(* PLC project mtcs_services, Institute of Astronomy OntoManager 0.0.1 *)
(* stored: creationDateTime 2024-08-13T09:12:25.681669, modificationDateTime 2024-08-13T09:12:25.681669 *)

TYPE ServicesTimingTimeSource : (LOCAL_CLOCK := 0, PTP_IEEE_1588 := 1);
END_TYPE

TYPE ServicesMeteoId : (WIND_SPEED_MINIMUM := 0, WIND_SPEED_AVERAGE := 1, WIND_SPEED_MAXIMUM := 2, WIND_DIRECTION_MINIMUM := 3, WIND_DIRECTION_AVERAGE := 4, WIND_DIRECTION_MAXIMUM := 5, AIR_PRESSURE := 6, AIR_TEMPERATURE := 7, INTERNAL_TEMPERATURE := 8, RELATIVE_HUMIDITY := 9, RAIN_ACCUMULATION := 10, RAIN_DURATION := 11, RAIN_INTENSITY := 12, RAIN_PEAK_INTENSITY := 13, HAIL_ACCUMULATION := 14, HAIL_DURATION := 15, HAIL_PEAK_INTENSITY := 16, HAIL_INTENSITY := 17, HEATING_TEMPERATURE := 18, HEATING_VOLTAGE := 19, SUPPLY_VOLTAGE := 20, REFERENCE_VOLTAGE := 21);
END_TYPE

TYPE ServicesParts : STRUCT
  timing : ServicesTiming;  (* Timing service *)
  meteo : ServicesMeteo;  (* Meteo service *)
  west : ServicesWest;  (* West service *)
  chiller : ServicesChiller;  (* Chiller service *)
  io : ServicesIO;  (* I/O modules *)
  configManager : ConfigManager;  (* The config manager (to load/save/activate configuration data) *)
END_STRUCT;
END_TYPE

TYPE ServicesTimingParts : STRUCT
  serialInfo : ServicesTimingSerialInfo;  (* Info acquired by serial link *)
END_STRUCT;
END_TYPE

TYPE ServicesWestParts : STRUCT
  bus : ModbusRTUBus;  (* The shared Modbus RTU bus *)
  domeTemperature : ServicesWestController;  (* The West coparts.chillerMainController.parts.chillerMainControllerntroller at the dome to control the temperature *)
  firstFloorTemperature : ServicesWestController;  (* The West controller at the first floor to control the temperature *)
  pumpsRoomTemperature : ServicesWestController;  (* The West controller at the pumps room to control the temperature *)
  oilHeatExchangerTemperature : ServicesWestController;  (* The West controller at the heat exchanger to control the oil temperature *)
  serversRoomTemperature : ServicesWestController;  (* The West controller at the servers room to control the temperature *)
END_STRUCT;
END_TYPE

TYPE ServicesChillerParts : STRUCT
  bus : ModbusRTUBus;  (* The shared Modbus RTU bus *)
  chillerMainController : ServicesChillerController;  (* The Chiller controller to control the water temperature *)
END_STRUCT;
END_TYPE

TYPE ServicesIOParts : STRUCT
  coupler : EtherCatDevice;  (* Coupler *)
  slot1 : EtherCatDevice;  (* Slot 1 *)
  slot2 : EtherCatDevice;  (* Slot 2 *)
  slot3 : EtherCatDevice;  (* Slot 3 *)
  slot4 : EtherCatDevice;  (* Slot 4 *)
END_STRUCT;
END_TYPE

TYPE ServicesProcesses : STRUCT
  initialize : Process;  (* Start initializing *)
  lock : Process;  (* Lock the system *)
  unlock : Process;  (* Unlock the system *)
  changeOperatingState : ChangeOperatingStateProcess;  (* Change the operating state (e.g. AUTO, MANUAL, ...) *)
END_STRUCT;
END_TYPE

TYPE ServicesTimingProcesses : STRUCT

END_STRUCT;
END_TYPE

TYPE ServicesMeteoProcesses : STRUCT

END_STRUCT;
END_TYPE

TYPE ServicesWestControllerProcesses : STRUCT
  updateProcessVariables : Process;  (* Read process variables *)
  updateConfigVariables : Process;  (* Read config variables *)
  writeSetpoint : ChangeSetpointProcess;  (* Write the setpoint *)
  writeOffset : ChangeParameterProcess;  (* Set an internal offset to Process Value *)
  writeProportinalBand : ChangeParameterProcess;  (* Set the Proportinal band constant *)
  writeResetTime : ChangeParameterProcess;  (* Set the Integral time constant *)
  writeRate : ChangeParameterProcess;  (* Set the Derivative time constant *)
  switchToManual : Process;  (* Switch controller to Manual *)
  switchToAuto : Process;  (* Switch controller to Auto *)
  writeOutputPower : ChangeParameterProcess;  (* Set a specific output power *)
  writeConfigToController : Process;  (* Write saved config to Controller *)
END_STRUCT;
END_TYPE

TYPE ServicesWestProcesses : STRUCT
  changeOperatingState : ChangeOperatingStateProcess;  (* Change the operating state (e.g. AUTO, MANUAL, ...) *)
END_STRUCT;
END_TYPE

TYPE ServicesChillerControllerProcesses : STRUCT
  updateConfigVariables : Process;  (* Read the Config variables *)
  updateMeasureVariables : Process;  (* Read the Measurement variables *)
  updateAlarmRegisters : Process;  (* Read the Alarm registers *)
  writeSetpoint : ChangeSetpointProcess;  (* Write the setpoint *)
  switchChillerON : Process;  (* Switch ON the Chiller *)
  switchChillerOFF : Process;  (* Switch OFF the Chiller *)
  resetUnitController : Process;  (* Reset Unit controller of the Chiller *)
  resetAlarms : Process;  (* Reset all activated alarms *)
END_STRUCT;
END_TYPE

TYPE ServicesChillerProcesses : STRUCT
  changeOperatingState : ChangeOperatingStateProcess;  (* Change the operating state (e.g. AUTO, MANUAL, ...) *)
END_STRUCT;
END_TYPE

TYPE ServicesStatuses : STRUCT
  initializationStatus : InitializationStatus;
  healthStatus : HealthStatus;
  busyStatus : BusyStatus;
  operatingStatus : OperatingStatus;
END_STRUCT;
END_TYPE

TYPE ServicesTimingStatuses : STRUCT
  healthStatus : HealthStatus;
END_STRUCT;
END_TYPE

TYPE ServicesTimingSerialInfoStatuses : STRUCT
  portHealthStatus : HealthStatus;
  transmissionHealthStatus : HealthStatus;
  checksumHealthStatus : HealthStatus;
  healthStatus : HealthStatus;
END_STRUCT;
END_TYPE

TYPE ServicesMeteoMeasurementStatuses : STRUCT
  enabledStatus : EnabledStatus;  (* Is the temperature being measured? *)
  healthStatus : HealthStatus;  (* Is the data valid and within range? *)
  alarmStatus : HiHiLoLoAlarmStatus;  (* Alarm status *)
END_STRUCT;
END_TYPE

TYPE ServicesMeteoStatuses : STRUCT
  meteoHealthStatus : HealthStatus;
  healthStatus : HealthStatus;
END_STRUCT;
END_TYPE

TYPE ServicesWestControllerStatuses : STRUCT
  healthStatus : HealthStatus;  (* Is the data valid and within range? *)
  alarmStatus : HiHiLoLoAlarmStatus;  (* Alarm status *)
END_STRUCT;
END_TYPE

TYPE ServicesWestStatuses : STRUCT
  healthStatus : HealthStatus;  (* Are the WESTs in healthy state (good) or not (bad) *)
  operatingStatus : OperatingStatus;  (* Are the WESTs being polled (auto) or not (manual)? *)
END_STRUCT;
END_TYPE

TYPE ServicesChillerControllerStatuses : STRUCT
  healthStatus : HealthStatus;  (* Is the data valid and within range? *)
  alarmStatusWatertemperature : HiHiLoLoAlarmStatus;  (* Alarm status about Water temperature *)
  alarmStatusWaterPumpSupervisor : HiHiLoLoAlarmStatus;  (* Alarm status about WaterPump supervisor *)
END_STRUCT;
END_TYPE

TYPE ServicesChillerStatuses : STRUCT
  healthStatus : HealthStatus;  (* Is the Chiller in healthy state (good) or not (bad) *)
  operatingStatus : OperatingStatus;  (* Is the Chiller being polled (auto) or not (manual)? *)
END_STRUCT;
END_TYPE

TYPE ServicesIOStatuses : STRUCT
  healthStatus : HealthStatus;  (* Is the I/O in a healthy state? *)
END_STRUCT;
END_TYPE

TYPE ServicesTimingConfig : STRUCT
  leapSeconds : INT;  (* Number of leap seconds, so that UTC = TAI + this value. See ftp://maia.usno.navy.mil/ser7/tai-utc.dat for the latest number. *)
  dut : LREAL;  (* Delta UT (= UT1 - UTC). Put to 0.0 to ignore. *)
  alwaysUseLocalClock : BOOL;  (* If TRUE, then the local clock (source=LOCAL_CLOCK) will be used even if an external (more accurate!) clock is available *)
  ignoreSerialError : BOOL;  (* Don't show the Servicestiming status as ERROR in case the serial link fails *)
END_STRUCT;
END_TYPE

TYPE ServicesMeteoConfig : STRUCT
  enableWeatherMonitoring : BOOL;  (* Enable weather monitoring and emergency closing *)
  wetLimit : LREAL;  (* Wet if (rainIntensity+hailIntrelaensity)>wetLimit *)
  windSpeedMinimum : MeasurementConfig;  (* Config for the wind speed minimum *)
  windSpeedAverage : MeasurementConfig;  (* Config for the wind speed average *)
  windSpeedMaximum : MeasurementConfig;  (* Config for the wind speed maximum *)
  windDirectionMinimum : MeasurementConfig;  (* Config for the wind direction minimum *)
  windDirectionAverage : MeasurementConfig;  (* Config for the wind direction average *)
  windDirectionMaximum : MeasurementConfig;  (* Config for the wind direction maximum *)
  airPressure : MeasurementConfig;  (* Config for the air pressure *)
  airTemperature : MeasurementConfig;  (* Config for the air temperature *)
  internalTemperature : MeasurementConfig;  (* Config for the internal temperature *)
  relativeHumidity : MeasurementConfig;  (* Config for the relative humidity *)
  rainAccumulation : MeasurementConfig;  (* Config for the rain accumulation *)
  rainDuration : MeasurementConfig;  (* Config for the rain duration *)
  rainIntensity : MeasurementConfig;  (* Config for the rain intensity *)
  rainPeakIntensity : MeasurementConfig;  (* Config for the rain peak intensity *)
  hailAccumulation : MeasurementConfig;  (* Config for the hail accumulation *)
  hailDuration : MeasurementConfig;  (* Config for the hail duration *)
  hailIntensity : MeasurementConfig;  (* Config for the hail intensity *)
  hailPeakIntensity : MeasurementConfig;  (* Config for the hail peak intensity *)
  heatingTemperature : MeasurementConfig;  (* Config for the heating temperature *)
  heatingVoltage : MeasurementConfig;  (* Config for the heating voltage *)
  supplyVoltage : MeasurementConfig;  (* Config for the supply voltage *)
  referenceVoltage : MeasurementConfig;  (* Config for the 3.5 V reference voltage *)
END_STRUCT;
END_TYPE

TYPE ServicesWestTemperatureTimeConfig : STRUCT
  enable : BOOL;  (* Enable this time (TRUE) or not (FALSE) *)
  hour : LREAL;  (* The time to change the setpoint, as decimal hour (e.g. 9.5 = 9:30 am) *)
  offset : LREAL;  (* Setpoint = air temperature of meteo station + this offset (in degrees celsius) *)
END_STRUCT;
END_TYPE

TYPE ServicesWestTemperatureUpdateConfig : STRUCT
  time0 : ServicesWestTemperatureTimeConfig;  (* Time config 0 *)
  time1 : ServicesWestTemperatureTimeConfig;  (* Time config 1 *)
  time2 : ServicesWestTemperatureTimeConfig;  (* Time config 2 *)
  time3 : ServicesWestTemperatureTimeConfig;  (* Time config 3 *)
  time4 : ServicesWestTemperatureTimeConfig;  (* Time config 4 *)
END_STRUCT;
END_TYPE

TYPE ServicesWestParametersAddressesConfig : STRUCT
  communicationWriteStatus : UINT := 1;  (* Communication Write Status *)
  manualControl : UINT := 2;  (* Manual control *)
  selfTune : UINT := 3;  (* Activate SelfTune *)
  preTune : UINT := 4;  (* Activate PreTune *)
  alarm1Status : UINT := 5;  (* Alarm 1 status *)
  alarm2Status : UINT := 6;  (* Alarm 2 status *)
  setpointRampling : UINT := 7;  (* Setpoint ramping *)
  loopAlarmStatus : UINT := 10;  (* Loop alarm status *)
  loopAlarm : UINT := 12;  (* Loop alarm *)
  digitalInput2 : UINT := 13;  (* State Option B digital input *)
  processVariable : UINT := 1;  (* Process Variable *)
  setpoint : UINT := 2;  (* Setpoint *)
  outputPower : UINT := 3;  (* Power percentage *)
  desviation : UINT := 4;  (* Difference ProcessVariable and Setpoint *)
  primaryProportionalBand : UINT := 6;  (* Primary Proportional band PB *)
  directActing : UINT := 7;  (* Direct reverse acting *)
  resetTime : UINT := 8;  (* Reset Time. Integral time constant *)
  rate : UINT := 9;  (* Rate. Derivative time constant *)
  output1ClycleTime : UINT := 10;  (* Output 1 cycle time in seconds *)
  scaleRangeLowerLimit : UINT := 11;  (* Lower Limit of input range *)
  scaleRangeUpperLimit : UINT := 12;  (* Upper Limit of input range *)
  alarm1Value : UINT := 13;  (* Alarm 1 active at this level *)
  alarm2Value : UINT := 14;  (* Alarm 2 active at this level *)
  manualReset : UINT := 15;  (* Bias value in percentage *)
  deadbandOverlap : UINT := 16;  (* Deadband and Overlap percentage *)
  onOffDiferential : UINT := 17;  (* Input span for ON/OFF differential *)
  decimalPointPosition : UINT := 18;  (* Decimal point position *)
  output2ClycleTime : UINT := 19;  (* Output 2 cycle time in seconds *)
  primaryOutputPowerLimit : UINT := 20;  (* Safety power limit in porcentage *)
  actualSetpoint : UINT := 21;  (* Current Setpoint value (ramping) *)
  setpointUpperLimit : UINT := 22;  (* Setpoint upper limit *)
  setpointLowerLimit : UINT := 23;  (* Setpoint lower limit *)
  setpointRampRate : UINT := 24;  (* Setpoint ramp rate *)
  inputFilterTimeContant : UINT := 25;  (* Input Filter time contant *)
  processValueOffset : UINT := 26;  (* Process Value offset *)
  alarm1Hysteresis : UINT := 32;  (* Alarm 1 hysteresis in percentage *)
  alarm2Hysteresis : UINT := 33;  (* Alarm 2 hysteresis in percentage *)
END_STRUCT;
END_TYPE

TYPE ServicesWestControllerVariables : STRUCT
  setpoint : LREAL;  (* Setpoint *)
  defaultSetpoint : LREAL;  (* Default setpoint *)
  minSetpoint : LREAL;  (* Minimun setpoint *)
  maxSetpoint : LREAL;  (* Maximal setpoint *)
  processValueOffset : LREAL;  (* Offset process varible *)
  differentialOnOff : LREAL;  (* On/Off differential *)
  alarmValue : LREAL;  (* Alarm value *)
  inputFilterTimeConstant : LREAL;  (* Input filter time constant *)
  cycleTime : LREAL;  (* Cycle time for control loop *)
  proportionalBand : UINT;  (* Proportional constant *)
  resetTime : UINT;  (* Integral time constant *)
  rate : UINT;  (* Dervative time constant *)
END_STRUCT;
END_TYPE

TYPE ServicesWestControllerConfig : STRUCT
  unitID : USINT;  (* The address or UnitID of the controller *)
  update : BOOL;  (* True to automatically update the setpoint *)
  warningMessage : STRING;  (* A warning message (empty = not shown) *)
  measurement : MeasurementConfig;  (* The measurement config *)
  variables : ServicesWestControllerVariables;  (* Configuration parameters *)
END_STRUCT;
END_TYPE

TYPE ServicesWestConfig : STRUCT
  updateProcessVariables : BOOL;  (* True to automatically update process variables *)
  updateVariablesPollingInterval : LREAL;  (* Time between bus reads in seconds *)
  domeTempControl : BOOL;  (* True to automatically update dome temperatures *)
  domeTempCycleTime : LREAL;  (* Time between bus checks in seconds *)
  hydraulicsTempControl : BOOL;  (* True to enable PID controller for hydraulics temperatures *)
  hydraulicsTempCycleTime : LREAL;  (* Cycle time for PID Controller in seconds *)
  hydraulicsProportionalConstantKP : LREAL;  (* Proportional constant (Kp) for PID Controller *)
  hydraulicsIntegralConstantTn : LREAL;  (* Integral constant (Tn) for PID Controller in seconds *)
  domeTemperature : ServicesWestControllerConfig;  (* The address of the Dome temperature controller *)
  firstFloorTemperature : ServicesWestControllerConfig;  (* The address of the first floor temperature controller *)
  pumpsRoomTemperature : ServicesWestControllerConfig;  (* The address of the pumps room temperature controller *)
  oilHeatExchangerTemperature : ServicesWestControllerConfig;  (* The address of the oil heat exchanger temperature controller *)
  serversRoomTemperature : ServicesWestControllerConfig;  (* The address of the servers room temperature controller *)
  parameterAddresses : ServicesWestParametersAddressesConfig;  (* Config about Modbus parameters addresses *)
  temperatureUpdate : ServicesWestTemperatureUpdateConfig;  (* The config for the temperature setpoint *)
END_STRUCT;
END_TYPE

TYPE ServicesChillerControllerParameterAddresses : STRUCT
  waterTankTemperature : UINT := 258;  (* Water tank temperature *)
  highPressureCircuit1 : UINT := 260;  (* High pressure of circuit 1 *)
  highPressureCircuit2 : UINT := 262;  (* High pressure of circuit 2 *)
  chillerCurrentInput : UINT := 264;  (* Chiller current input *)
  waterPumpCurrentInput : UINT := 266;  (* Water pump current input *)
  evaporatorOutTemp1 : UINT := 268;  (* Evaporator out temperature 1 *)
  evaporatorOutTemp2 : UINT := 270;  (* Evaporator out temperature 2 *)
  ambientTemperature : UINT := 272;  (* Ambient temperature *)
  waterPumpChassisTemp : UINT := 274;  (* Water Pump chassis temperature *)
  digitalInputStatus1 : UINT := 512;  (* Flow switch status *)
  digitalInputStatus2 : UINT := 513;  (* Digital input status 2 *)
  digitalInputStatus3 : UINT := 514;  (* Digital input status 3 *)
  digitalInputStatus4 : UINT := 515;  (* Digital input status 4 *)
  setpoint : UINT := 768;  (* Setpoint parameter address *)
  minSetpoint : UINT := 769;  (* Minimal Setpoint parameter address *)
  maxSetpoint : UINT := 770;  (* Maximal Setpoint parameter address *)
  trippingBand : UINT := 774;  (* Tripping Band parameter address *)
  unitStatus : UINT := 1280;  (* Unit Status parameter address *)
  unitControllerReset : UINT := 1282;  (* Unit Controlelr reset parameter address *)
  relayOutputStatus1 : UINT := 2048;  (* Relay output status 1 *)
  relayOutputStatus2 : UINT := 2049;  (* Relay output status 2 *)
  relayOutputStatus3 : UINT := 2050;  (* Relay output status 3 *)
  relayOutputStatus4 : UINT := 2051;  (* Relay output status 4 *)
  relayOutputStatus5 : UINT := 2052;  (* Relay output status 5 *)
  relayOutputStatus6 : UINT := 2053;  (* Relay output status 6 *)
  relayOutputStatus7 : UINT := 2054;  (* Relay output status 7 *)
  AnalogOutputStatus1 : UINT := 2304;  (* Fan Condenser1 Output *)
  AnalogOutputStatus2 : UINT := 2306;  (* Fan Condenser2 Output *)
  alarmStatus1 : UINT := 3328;  (* Alarm status 1 *)
  alarmStatus2 : UINT := 3329;  (* Alarm status 2 *)
  alarmStatus3 : UINT := 3330;  (* Alarm status 3 *)
  alarmStatus6 : UINT := 3333;  (* Alarm status 6 *)
  alarmStatus7 : UINT := 3334;  (* Alarm status 7 *)
  alarmStatus10 : UINT := 3337;  (* Alarm status 10 *)
  alarmStatus11 : UINT := 3338;  (* Alarm status 11 *)
  hoursCompressor1 : UINT := 3584;  (* Operation hours of compressor 1 *)
  hoursCompressor2 : UINT := 3585;  (* Operation hours of compressor 2 *)
  hoursCompressor3 : UINT := 3586;  (* Operation hours of compressor 3 *)
  hoursCompressor4 : UINT := 3587;  (* Operation hours of compressor 4 *)
  hoursPump : UINT := 3590;  (* Operation hours of water pump *)
  alarmOilCompressor1 : UINT := 3840;  (* Alarm oil Compressor 1 *)
  alarmOilCompressor2 : UINT := 3841;  (* Alarm oil Compressor 2 *)
  alarmOilCompressor3 : UINT := 3842;  (* Alarm oil Compressor 3 *)
  alarmOilCompressor4 : UINT := 3843;  (* Alarm oil Compressor 4 *)
  alarmFanOverload : UINT := 3846;  (* Alarm fan overload *)
  alarmColdSideFlowSwitch : UINT := 3847;  (* Alarm cold side flow switch *)
  alarmHotSideFlowSwitch : UINT := 3848;  (* Alarm hot side flow switch *)
  alarmCirc1LowTempPressDI : UINT := 3849;  (* Alarm circuit 1 low temppress DI *)
  alarmCirc2LowTempPressDI : UINT := 3850;  (* Alarm circuit 2 low temppress DI *)
  alarmCirc1LowTempPressPB : UINT := 3851;  (* Alarm circuit 1 low temppress PB *)
  alarmCirc2LowTempPressPB : UINT := 3852;  (* Alarm circuit 2 low temppress PB *)
END_STRUCT;
END_TYPE

TYPE ServicesChillerControllerAlarmStatus1 : STRUCT
  bit0 : STRING := 'PROBE8 (EVAP2. WATER TEMPERATURE)';
  bit1 : STRING := 'PROBE9 (AMBIENT TEMPERATURE)';
  bit2 : STRING := 'PROBE10 (NOT USED)';
  bit3 : STRING := 'PROBE11 (NOT USED)';
  bit4 : STRING := 'PROBE12 (NOT USED)';
  bit5 : STRING := 'COMPRESSOR1 MAINTENANCE';
  bit6 : STRING := 'COMPRESSOR2 MAINTENANCE';
  bit7 : STRING := 'COMPRESSOR3 MAINTENANCE';
  bit8 : STRING := 'ALARM NOT DEFINED';
  bit9 : STRING := 'PROBE1 (NOT USED)';
  bit10 : STRING := 'PROBE2 (TANK. WATER TEMPERATURE)';
  bit11 : STRING := 'PROBE3 (HIGH PRESSURE CRIC1)';
  bit12 : STRING := 'PROBE4 (HIGH PRESSURE CRIC2)';
  bit13 : STRING := 'PROBE5 (NOT USED)';
  bit14 : STRING := 'PROBE6 (NOT USED)';
  bit15 : STRING := 'PROBE7 (EVAP1. WATER TEMPERATURE)';
END_STRUCT;
END_TYPE

TYPE ServicesChillerControllerAlarmStatus2 : STRUCT
  bit0 : STRING := 'ALARM NOT DEFINED';
  bit1 : STRING := 'ALARM NOT DEFINED';
  bit2 : STRING := 'ALARM NOT DEFINED';
  bit3 : STRING := 'ALARM NOT DEFINED';
  bit4 : STRING := 'ALARM NOT DEFINED';
  bit5 : STRING := 'ALARM NOT DEFINED';
  bit6 : STRING := 'ALARM NOT DEFINED';
  bit7 : STRING := 'ALARM NOT DEFINED';
  bit8 : STRING := 'COMPRESSOR4 MAINTENANCE';
  bit9 : STRING := 'ALARM NOT DEFINED';
  bit10 : STRING := 'ALARM NOT DEFINED';
  bit11 : STRING := 'PUMP/DELIVERY FAN MAINTENANCE';
  bit12 : STRING := 'EVAPORATOR2 PUMP MAINTENANCE';
  bit13 : STRING := 'CONDENSER1 PUMP MAINTENANCE';
  bit14 : STRING := 'CONDENSER2 PUMP MAINTENANCE';
  bit15 : STRING := 'ALARM NOT DEFINED';
END_STRUCT;
END_TYPE

TYPE ServicesChillerControllerAlarmStatus3 : STRUCT
  bit0 : STRING := 'ALARM NOT DEFINED';
  bit1 : STRING := 'ALARM NOT DEFINED';
  bit2 : STRING := 'ALARM NOT DEFINED';
  bit3 : STRING := 'ALARM NOT DEFINED';
  bit4 : STRING := 'ALARM NOT DEFINED';
  bit5 : STRING := 'ALARM NOT DEFINED';
  bit6 : STRING := 'ALARM NOT DEFINED';
  bit7 : STRING := 'ALARM NOT DEFINED';
  bit8 : STRING := 'CIRCUIT1 DEFROST';
  bit9 : STRING := 'CIRCUIT2 DEFROST';
  bit10 : STRING := 'NETWORK FREQUENCY';
  bit11 : STRING := 'LOW INLET AIR TEMPERATURE';
  bit12 : STRING := 'ALARM NOT DEFINED';
  bit13 : STRING := 'ALARM NOT DEFINED';
  bit14 : STRING := 'EVAPORATOR LOW OUTLET TEMPERATURE';
  bit15 : STRING := 'EVAPORATOR HIGH OUTLET TEMPERATURE';
END_STRUCT;
END_TYPE

TYPE ServicesChillerControllerAlarmStatus6 : STRUCT
  bit0 : STRING := 'COMPRESSOR1 THERMAL OVERLOAD';
  bit1 : STRING := 'COMPRESSOR2 THERMAL OVERLOAD';
  bit2 : STRING := 'COMPRESSOR3 THERMAL OVERLOAD';
  bit3 : STRING := 'COMPRESSOR4 THERMAL OVERLOAD';
  bit4 : STRING := 'ALARM NOT DEFINED';
  bit5 : STRING := 'ALARM NOT DEFINED';
  bit6 : STRING := 'CIRC1 COND. FAN THERMAL OVERLOAD';
  bit7 : STRING := 'CIRC2 COND. FAN THERMAL OVERLOAD';
  bit8 : STRING := 'ALARM NOT DEFINED';
  bit9 : STRING := 'ALARM NOT DEFINED';
  bit10 : STRING := 'COMPRESSOR1 HIGH PRESSURE';
  bit11 : STRING := 'COMPRESSOR2 HIGH PRESSURE';
  bit12 : STRING := 'COMPRESSOR3 HIGH PRESSURE';
  bit13 : STRING := 'COMPRESSOR4 HIGH PRESSURE';
  bit14 : STRING := 'ALARM NOT DEFINED';
  bit15 : STRING := 'ALARM NOT DEFINED';
END_STRUCT;
END_TYPE

TYPE ServicesChillerControllerAlarmStatus7 : STRUCT
  bit0 : STRING := 'ALARM NOT DEFINED';
  bit1 : STRING := 'ALARM NOT DEFINED';
  bit2 : STRING := 'ALARM NOT DEFINED';
  bit3 : STRING := 'ALARM NOT DEFINED';
  bit4 : STRING := 'ALARM NOT DEFINED';
  bit5 : STRING := 'ALARM NOT DEFINED';
  bit6 : STRING := 'ALARM NOT DEFINED';
  bit7 : STRING := 'ALARM NOT DEFINED';
  bit8 : STRING := 'EVAP1 WATER PUMP THERMAL OVERLOAD';
  bit9 : STRING := 'EVAP2 WATER PUMP THERMAL OVERLOAD';
  bit10 : STRING := 'COND1 PUMP THERMAL OVERLOAD';
  bit11 : STRING := 'COND2 PUMP THERMAL OVERLOAD';
  bit12 : STRING := 'CIRC1 HIGH PRESSURE SWITCH TRIPPED';
  bit13 : STRING := 'CIRC2 HIGH PRESSURE SWITCH TRIPPED';
  bit14 : STRING := 'CIRC1 HIGH PRESSURE PROBE';
  bit15 : STRING := 'CIRC2 HIGH PRESSURE PROBE';
END_STRUCT;
END_TYPE

TYPE ServicesChillerControllerAlarmStatus10 : STRUCT
  bit0 : STRING := 'HOT SIDE FLOW SWITCH';
  bit1 : STRING := 'CIC1 LOW PRESSURE SWITCH';
  bit2 : STRING := 'CIC2 LOW PRESSURE SWITCH';
  bit3 : STRING := 'CIC1 LOW PRESSURE PROBE';
  bit4 : STRING := 'CIC2 LOW PRESSURE PROBE';
  bit5 : STRING := 'CIRC1 PUMP-DOWN AT STARTUP';
  bit6 : STRING := 'CIRC2 PUMP-DOWN AT STARTUP';
  bit7 : STRING := 'CIRC1 PUMP-DOWN AT SHUTDOWN';
  bit8 : STRING := 'COMPRESSOR1 OIL';
  bit9 : STRING := 'COMPRESSOR2 OIL';
  bit10 : STRING := 'COMPRESSOR3 OIL';
  bit11 : STRING := 'COMPRESSOR4 OIL';
  bit12 : STRING := 'ALARM NOT DEFINED';
  bit13 : STRING := 'ALARM NOT DEFINED';
  bit14 : STRING := 'DELIVERY FAN THERMAL OVERLOAD';
  bit15 : STRING := 'COLD SIDE FLOW SWITCH';
END_STRUCT;
END_TYPE

TYPE ServicesChillerControllerAlarmStatus11 : STRUCT
  bit0 : STRING := 'COMPRESSOR4 DISCHARGE HIGH TEMPERATURE';
  bit1 : STRING := 'ALARM NOT DEFINED';
  bit2 : STRING := 'ALARM NOT DEFINED';
  bit3 : STRING := 'GENERAL ALARM FROM DIGITAL INPUT';
  bit4 : STRING := 'ALARM NOT DEFINED';
  bit5 : STRING := 'ALARM NOT DEFINED';
  bit6 : STRING := 'ALARM NOT DEFINED';
  bit7 : STRING := 'ALARM NOT DEFINED';
  bit8 : STRING := 'CIRC2 PUMP-DOWN AT SHUTDOWN';
  bit9 : STRING := 'CIRC1 CHILLER ANTI-FREEZE';
  bit10 : STRING := 'CIRC2 CHILLER ANTI-FREEZE';
  bit11 : STRING := 'CIRC1 PUMP ANTI-FREEZE';
  bit12 : STRING := 'CIRC2 PUMP ANTI-FREEZE';
  bit13 : STRING := 'COMPRESSOR1 DISCHARGE HIGH TEMPERATURE';
  bit14 : STRING := 'COMPRESSOR2 DISCHARGE HIGH TEMPERATURE';
  bit15 : STRING := 'COMPRESSOR3 DISCHARGE HIGH TEMPERATURE';
END_STRUCT;
END_TYPE

TYPE ServicesChillerControllerBitwiseConfig : STRUCT
  statusOnMask : UINT := 768;  (* Word check if Chiller is ON *)
  switchOnMask : UINT := 1028;  (* Word to switch ON the Chiller *)
  switchOffMask : UINT := 1;  (* Word to switch OFF the Chiller *)
  resetUnitMask : UINT := 128;  (* Word to reset controller Unit *)
  resetAlarmMask : UINT := 4112;  (* Word to reset Alarm *)
  flowSwitchMask : UINT := 2048;  (* Word to check if Flow switch is ON *)
  alarmOnMask : UINT := 257;  (* Word to check if Alarm relay is ON *)
  waterPumpOnMask : UINT := 514;  (* Word to check if water Pump relay is ON *)
  compressor1Mask : UINT := 8224;  (* Word to check if Compressor1 is ON *)
  compressor2Mask : UINT := 4112;  (* Word to check if Compressor2 is ON *)
  compressor3Mask : UINT := 2056;  (* Word to check if Compressor3 is ON *)
  compressor4Mask : UINT := 1028;  (* Word to check if Compressor4 is ON *)
  bit0 : UINT := 1;  (* Word mask to check bit0 *)
  bit1 : UINT := 2;  (* Word mask to check bit1 *)
  bit2 : UINT := 4;  (* Word mask to check bit2 *)
  bit3 : UINT := 8;  (* Word mask to check bit3 *)
  bit4 : UINT := 16;  (* Word mask to check bit4 *)
  bit5 : UINT := 32;  (* Word mask to check bit5 *)
  bit6 : UINT := 64;  (* Word mask to check bit6 *)
  bit7 : UINT := 128;  (* Word mask to check bit7 *)
  bit8 : UINT := 256;  (* Word mask to check bit8 *)
  bit9 : UINT := 512;  (* Word mask to check bit9 *)
  bit10 : UINT := 1024;  (* Word mask to check bit10 *)
  bit11 : UINT := 2048;  (* Word mask to check bit11 *)
  bit12 : UINT := 4096;  (* Word mask to check bit12 *)
  bit13 : UINT := 8192;  (* Word mask to check bit13 *)
  bit14 : UINT := 16384;  (* Word mask to check bit14 *)
  bit15 : UINT := 32768;  (* Word mask to check bit15 *)
END_STRUCT;
END_TYPE

TYPE ServicesChillerControllerAlarmStatusRegisters : STRUCT
  AlarmStatus1 : ServicesChillerControllerAlarmStatus1;  (* Alarm indicators at AlarmStatus1 register *)
  AlarmStatus2 : ServicesChillerControllerAlarmStatus2;  (* Alarm indicators at AlarmStatus2 register *)
  AlarmStatus3 : ServicesChillerControllerAlarmStatus3;  (* Alarm indicators at AlarmStatus3 register *)
  AlarmStatus6 : ServicesChillerControllerAlarmStatus6;  (* Alarm indicators at AlarmStatus6 register *)
  AlarmStatus7 : ServicesChillerControllerAlarmStatus7;  (* Alarm indicators at AlarmStatus7 register *)
  AlarmStatus10 : ServicesChillerControllerAlarmStatus10;  (* Alarm indicators at AlarmStatus10 register *)
  AlarmStatus11 : ServicesChillerControllerAlarmStatus11;  (* Alarm indicators at AlarmStatus11 register *)
END_STRUCT;
END_TYPE

TYPE ServicesChillerControllerVariables : STRUCT
  setpoint : LREAL;  (* Setpoint *)
  minSetpoint : LREAL;  (* Minimun setpoint *)
  maxSetpoint : LREAL;  (* Maximal setpoint *)
  trippingBand : LREAL;  (* Tripping band *)
END_STRUCT;
END_TYPE

TYPE ServicesChillerControllerConfig : STRUCT
  unitID : USINT;  (* The address or UnitID of the controller *)
  waterTankTemperatureMeasurement : MeasurementConfig;  (* The WaterTank measurement config *)
  warningMessageWaterTemperatureMeasurement : STRING;  (* A warning message (empty = not shown) *)
  waterPumpSupervisorMeasurement : MeasurementConfig;  (* The WaterPump supervisor measurement config *)
  messageWaterPumpSupervisorMeasurement : STRING;  (* A message to be shown on config tab *)
  warningMessageWaterPumpSupervisorMeasurement : STRING;  (* A warning message (empty = not shown) *)
  parameterAddresses : ServicesChillerControllerParameterAddresses;  (* Config about Modbus parameters addresses *)
  variables : ServicesChillerControllerVariables;  (* Config value for some parameters *)
  alarmRegisters : ServicesChillerControllerAlarmStatusRegisters;  (* Config about Alarm statuses registers *)
  bitwise : ServicesChillerControllerBitwiseConfig;  (* Config about words and masks for bitwise actions *)
END_STRUCT;
END_TYPE

TYPE ServicesChillerConfig : STRUCT
  updateSetpoint : BOOL;  (* True to automatically update the setpoint *)
  temperatureToChangeSetpoint : LREAL;  (* Temperature to change Setpoint *)
  summerSetpoint : LREAL;  (* Temperature setpoint for summer *)
  winterSetpoint : LREAL;  (* Temperature setpoint for winter *)
  offsetSetpoint : LREAL;  (* Setpoint = air temperature of meteo station + this offset (in degrees celsius) *)
  updateSetpointInterval : LREAL;  (* Time interval to check ambient/setpoint temperature in seconds *)
  updateVariables : BOOL;  (* True to automatically update the setpoint *)
  pollingMeasuresInterval : LREAL;  (* Time between bus measurement reads in seconds *)
  pollingConfigInterval : LREAL;  (* Time between bus config variables reads in seconds *)
  pollingAlarmsInterval : LREAL;  (* Time between bus alarm registers reads in seconds *)
  chillerMainController : ServicesChillerControllerConfig;  (* The Chiller controller config *)
END_STRUCT;
END_TYPE

TYPE ServicesConfig : STRUCT
  timing : ServicesTimingConfig;  (* Timing config *)
  meteo : ServicesMeteoConfig;  (* Meteo config *)
  west : ServicesWestConfig;  (* West config *)
  chiller : ServicesChillerConfig;  (* Chiller config *)
END_STRUCT;
END_TYPE

FUNCTION_BLOCK SM_Services
  VAR_INPUT
    {attribute 'OPC.UA.DA' := '1'}
    {attribute 'OPC.UA.DA.Access' := '1'}
    editableConfig : ServicesConfig;  (* Editable configuration of the Services subsystem *)
  END_VAR
  VAR_OUTPUT
    {attribute 'OPC.UA.DA' := '1'}
    {attribute 'OPC.UA.DA.Access' := '1'}
    actualStatus : STRING;  (* Current status description *)
    previousStatus : STRING;  (* Previous status description *)
    {attribute 'OPC.UA.DA' := '1'}
    {attribute 'OPC.UA.DA.Access' := '1'}
    config : ServicesConfig;  (* Active configuration of the Services subsystem *)
    statuses : ServicesStatuses;  (* Statuses of the state machine *)
    parts : ServicesParts;  (* Parts of the state machine *)
    processes : ServicesProcesses;  (* Processes of the state machine *)
  END_VAR
  VAR_IN_OUT
    {attribute 'OPC.UA.DA' := '0'}
    operatorStatus : OperatorStatus;  (* Shared operator status *)
    {attribute 'OPC.UA.DA' := '0'}
    domeApertureStatus : ApertureStatus;  (* Is the dome open or closed? *)
  END_VAR

            parts.timing(
    operatorStatus := operatorStatus,
    config := config.timing);
parts.meteo( config := config.meteo );
parts.west(
    operatorStatus := operatorStatus,
    config := config.west,
    airTemperature := parts.meteo.airTemperature,
    domeApertureStatus := domeApertureStatus);
parts.chiller(
    operatorStatus := operatorStatus,
    config := config.chiller,
    airTemperature := parts.meteo.airTemperature);
parts.io();
parts.configManager( isEnabled := operatorStatus.tech );
statuses.initializationStatus();
statuses.healthStatus(
    isGood := parts.timing.statuses.healthStatus.isGood AND (parts.meteo.statuses.healthStatus.isGood AND (parts.west.statuses.healthStatus.isGood AND (parts.chiller.statuses.healthStatus.isGood AND parts.io.statuses.healthStatus.isGood))),
    hasWarning := parts.timing.statuses.healthStatus.hasWarning OR (parts.meteo.statuses.healthStatus.hasWarning OR (parts.west.statuses.healthStatus.hasWarning OR (parts.chiller.statuses.healthStatus.hasWarning OR parts.io.statuses.healthStatus.hasWarning))));
statuses.busyStatus( isBusy := statuses.initializationStatus.initializing );
statuses.operatingStatus( superState := statuses.initializationStatus.initialized );
processes.initialize( isEnabled := statuses.initializationStatus.shutdown OR (statuses.initializationStatus.initializingFailed OR statuses.initializationStatus.initialized) );
processes.lock( isEnabled := operatorStatus.tech AND statuses.initializationStatus.initialized );
processes.unlock( isEnabled := operatorStatus.tech AND statuses.initializationStatus.locked );
processes.changeOperatingState( isEnabled := FALSE );

          

{attribute 'TcRpcEnable' := '1'}
METHOD initialize : RequestResults
                  initialize := THIS^.processes.initialize.request();

                
END_METHOD

{attribute 'TcRpcEnable' := '1'}
METHOD lock : RequestResults
                  lock := THIS^.processes.lock.request();

                
END_METHOD

{attribute 'TcRpcEnable' := '1'}
METHOD unlock : RequestResults
                  unlock := THIS^.processes.unlock.request();

                
END_METHOD

{attribute 'TcRpcEnable' := '1'}
METHOD changeOperatingState : RequestResults
  VAR_INPUT
    state : OperatingStates;
  END_VAR
                  changeOperatingState := THIS^.processes.changeOperatingState.request( state := state );

                
END_METHOD

{attribute 'TcRpcEnable' := '1'}
METHOD _log : BOOL
  VAR_INPUT
    name : STRING;  (* Name of this function block instance *)
  END_VAR
  VAR_IN_OUT
    buffer : LogBuffer;  (* Buffer to write all logging to *)
  END_VAR
  VAR
    subBuffer : LogBuffer;  (* Temporary buffer to write logging by parts (sub-statemachines) to *)
  END_VAR
                  THIS^.parts.timing._log(
    name := 'timing',
    buffer := subBuffer);
THIS^.parts.meteo._log(
    name := 'meteo',
    buffer := subBuffer);
THIS^.parts.west._log(
    name := 'west',
    buffer := subBuffer);
THIS^.parts.chiller._log(
    name := 'chiller',
    buffer := subBuffer);
THIS^.parts.io._log(
    name := 'io',
    buffer := subBuffer);
THIS^.parts.configManager._log(
    name := 'configManager',
    buffer := subBuffer);
THIS^.processes.initialize._log(
    name := 'processes.initialize',
    buffer := subBuffer);
THIS^.processes.lock._log(
    name := 'processes.lock',
    buffer := subBuffer);
THIS^.processes.unlock._log(
    name := 'processes.unlock',
    buffer := subBuffer);
THIS^.processes.changeOperatingState._log(
    name := 'processes.changeOperatingState',
    buffer := subBuffer);
LOGGER(
    name := name,
    actualStatus := THIS^.actualStatus,
    previousStatus := THIS^.previousStatus,
    buffer := buffer,
    subBuffer := subBuffer,
    pHealthStatus := ADR(THIS^.statuses.healthStatus),
    pBusyStatus := ADR(THIS^.statuses.busyStatus));

                
END_METHOD
END_FUNCTION_BLOCK

FUNCTION_BLOCK SM_ServicesTiming
  VAR_INPUT
    {attribute 'OPC.UA.DA' := '1'}
    {attribute 'OPC.UA.DA.Access' := '1'}
    fromEL6688 AT %I* : TmcFromIoEL6688;  (* Data from the EL6688 *)
    {attribute 'OPC.UA.DA' := '1'}
    {attribute 'OPC.UA.DA.Access' := '1'}
    fromEcatMaster AT %I* : TmcFromIoEcatMaster;  (* Data from the EtherCAT master *)
    {attribute 'OPC.UA.DA' := '1'}
    {attribute 'OPC.UA.DA.Access' := '1'}
    fromCppTiming AT %I* : TmcToPlcTiming;  (* Data from the C++ task *)
  END_VAR
  VAR_OUTPUT
    {attribute 'OPC.UA.DA' := '1'}
    {attribute 'OPC.UA.DA.Access' := '1'}
    actualStatus : STRING;  (* Current status description *)
    previousStatus : STRING;  (* Previous status description *)
    {attribute 'OPC.UA.DA' := '1'}
    {attribute 'OPC.UA.DA.Access' := '1'}
    toCppTiming AT %Q* : TmcFromPlcTiming;  (* Data to the C++ task *)
    {attribute 'OPC.UA.DA' := '1'}
    {attribute 'OPC.UA.DA.Access' := '1'}
    utcDateString : STRING;  (* UTC date as a string of format YYYY-MM-DD *)
    {attribute 'OPC.UA.DA' := '1'}
    {attribute 'OPC.UA.DA.Access' := '1'}
    utcTimeString : STRING;  (* UTC time as a string of format HH-MM-SS.SSS *)
    {attribute 'OPC.UA.DA' := '1'}
    {attribute 'OPC.UA.DA.Access' := '1'}
    internalTimestampString : STRING;  (* String representation of the internal timestamp *)
    {attribute 'OPC.UA.DA' := '1'}
    {attribute 'OPC.UA.DA.Access' := '1'}
    externalTimestampString : STRING;  (* String representation of the external timestamp (note: this is TAI, not UTC!) *)
    statuses : ServicesTimingStatuses;  (* Statuses of the state machine *)
    parts : ServicesTimingParts;  (* Parts of the state machine *)
    processes : ServicesTimingProcesses;  (* Processes of the state machine *)
  END_VAR
  VAR_IN_OUT
    {attribute 'OPC.UA.DA' := '0'}
    operatorStatus : OperatorStatus;  (* Shared operator status *)
    {attribute 'OPC.UA.DA' := '0'}
    config : ServicesTimingConfig;  (* The config *)
  END_VAR

            parts.serialInfo();
statuses.healthStatus( isGood := config.ignoreSerialError OR parts.serialInfo.statuses.healthStatus.good );

          

{attribute 'TcRpcEnable' := '1'}
METHOD _log : BOOL
  VAR_INPUT
    name : STRING;  (* Name of this function block instance *)
  END_VAR
  VAR_IN_OUT
    buffer : LogBuffer;  (* Buffer to write all logging to *)
  END_VAR
  VAR
    subBuffer : LogBuffer;  (* Temporary buffer to write logging by parts (sub-statemachines) to *)
  END_VAR
                  THIS^.parts.serialInfo._log(
    name := 'serialInfo',
    buffer := subBuffer);
LOGGER(
    name := name,
    actualStatus := THIS^.actualStatus,
    previousStatus := THIS^.previousStatus,
    buffer := buffer,
    subBuffer := subBuffer,
    pHealthStatus := ADR(THIS^.statuses.healthStatus));

                
END_METHOD
END_FUNCTION_BLOCK

FUNCTION_BLOCK SM_ServicesTimingSerialInfo
  VAR_OUTPUT
    {attribute 'OPC.UA.DA' := '1'}
    {attribute 'OPC.UA.DA.Access' := '1'}
    actualStatus : STRING;  (* Current status description *)
    previousStatus : STRING;  (* Previous status description *)
    {attribute 'OPC.UA.DA' := '1'}
    {attribute 'OPC.UA.DA.Access' := '1'}
    serialTimeout : BOOL;  (* Is the serial data not being received within time? *)
    {attribute 'OPC.UA.DA' := '1'}
    {attribute 'OPC.UA.DA.Access' := '1'}
    comError : BOOL;  (* Is there any problem with the COM port? *)
    {attribute 'OPC.UA.DA' := '1'}
    {attribute 'OPC.UA.DA.Access' := '1'}
    comErrorID : INT;  (* COM error id (see Beckhoff ComError_t) *)
    {attribute 'OPC.UA.DA' := '1'}
    {attribute 'OPC.UA.DA.Access' := '1'}
    comErrorDescription : STRING;  (* Description of the COM error id *)
    {attribute 'OPC.UA.DA' := '1'}
    {attribute 'OPC.UA.DA.Access' := '1'}
    time_h : USINT;  (* Time: hours (0-24) *)
    {attribute 'OPC.UA.DA' := '1'}
    {attribute 'OPC.UA.DA.Access' := '1'}
    time_m : USINT;  (* Time: minutes (0-59) *)
    {attribute 'OPC.UA.DA' := '1'}
    {attribute 'OPC.UA.DA.Access' := '1'}
    time_s : USINT;  (* Time: seconds (0-59, or 60 if leap second) *)
    {attribute 'OPC.UA.DA' := '1'}
    {attribute 'OPC.UA.DA.Access' := '1'}
    latitude_deg : USINT;  (* Latitude: degrees (0-90) *)
    {attribute 'OPC.UA.DA' := '1'}
    {attribute 'OPC.UA.DA.Access' := '1'}
    latitude_min : REAL;  (* Latitude: minutes (0.0-59.99999) *)
    {attribute 'OPC.UA.DA' := '1'}
    {attribute 'OPC.UA.DA.Access' := '1'}
    latitude_sign : STRING;  (* Latitude: sign (either 'N' or 'S') *)
    {attribute 'OPC.UA.DA' := '1'}
    {attribute 'OPC.UA.DA.Access' := '1'}
    longitude_deg : USINT;  (* Longitude: degrees (0-180) *)
    {attribute 'OPC.UA.DA' := '1'}
    {attribute 'OPC.UA.DA.Access' := '1'}
    longitude_min : REAL;  (* Longitude: minutes (0.0-59.99999) *)
    {attribute 'OPC.UA.DA' := '1'}
    {attribute 'OPC.UA.DA.Access' := '1'}
    longitude_sign : STRING;  (* Longitude: sign (either 'E' or 'W') *)
    {attribute 'OPC.UA.DA' := '1'}
    {attribute 'OPC.UA.DA.Access' := '1'}
    positionFix : BOOL;  (* True if a position fix was accomplished, False if not *)
    {attribute 'OPC.UA.DA' := '1'}
    {attribute 'OPC.UA.DA.Access' := '1'}
    satellitesUsed : USINT;  (* Number of satellites used *)
    {attribute 'OPC.UA.DA' := '1'}
    {attribute 'OPC.UA.DA.Access' := '1'}
    horizontalDilutionOfPosition : REAL;  (* Horizontal dilution of position *)
    {attribute 'OPC.UA.DA' := '1'}
    {attribute 'OPC.UA.DA.Access' := '1'}
    meanSeaLevelAltitude : REAL;  (* Mean altitude above sea level in meters *)
    {attribute 'OPC.UA.DA' := '1'}
    {attribute 'OPC.UA.DA.Access' := '1'}
    geoidSeparation : REAL;  (* Geoid separation in meters *)
    {attribute 'OPC.UA.DA' := '1'}
    {attribute 'OPC.UA.DA.Access' := '1'}
    checksum : USINT;  (* Checksum send by the time server *)
    {attribute 'OPC.UA.DA' := '1'}
    {attribute 'OPC.UA.DA.Access' := '1'}
    calculatedChecksum : USINT;  (* Checksum calculated by the PLC *)
    statuses : ServicesTimingSerialInfoStatuses;  (* Statuses of the state machine *)
  END_VAR

            statuses.portHealthStatus( isGood := NOT(comError) );
statuses.transmissionHealthStatus( isGood := NOT(serialTimeout) );
statuses.checksumHealthStatus( isGood := checksum = calculatedChecksum );
statuses.healthStatus( isGood := statuses.portHealthStatus.good AND (statuses.transmissionHealthStatus.good AND statuses.checksumHealthStatus.good) );

          

{attribute 'TcRpcEnable' := '1'}
METHOD _log : BOOL
  VAR_INPUT
    name : STRING;  (* Name of this function block instance *)
  END_VAR
  VAR_IN_OUT
    buffer : LogBuffer;  (* Buffer to write all logging to *)
  END_VAR
  VAR
    subBuffer : LogBuffer;  (* Temporary buffer to write logging by parts (sub-statemachines) to *)
  END_VAR
                  LOGGER(
    name := name,
    actualStatus := THIS^.actualStatus,
    previousStatus := THIS^.previousStatus,
    buffer := buffer,
    subBuffer := subBuffer,
    pHealthStatus := ADR(THIS^.statuses.healthStatus));

                
END_METHOD
END_FUNCTION_BLOCK

FUNCTION_BLOCK SM_ServicesMeteoMeasurement
  VAR_INPUT
    {attribute 'OPC.UA.DA' := '1'}
    {attribute 'OPC.UA.DA.Access' := '1'}
    id : ServicesMeteoId;  (* ID *)
    {attribute 'OPC.UA.DA' := '0'}
    inputString : STRING;  (* Input string from the meteo station *)
  END_VAR
  VAR_OUTPUT
    {attribute 'OPC.UA.DA' := '1'}
    {attribute 'OPC.UA.DA.Access' := '1'}
    actualStatus : STRING;  (* Current status description *)
    previousStatus : STRING;  (* Previous status description *)
    {attribute 'OPC.UA.DA' := '1'}
    {attribute 'OPC.UA.DA.Access' := '1'}
    data : QuantityValue;  (* Actual value *)
    {attribute 'OPC.UA.DA' := '1'}
    {attribute 'OPC.UA.DA.Access' := '1'}
    invalidData : BOOL;  (* True if the data is invalid *)
    {attribute 'OPC.UA.DA' := '1'}
    {attribute 'OPC.UA.DA.Access' := '1'}
    lastChar : STRING;  (* Last character *)
    {attribute 'OPC.UA.DA' := '1'}
    {attribute 'OPC.UA.DA.Access' := '1'}
    name : STRING;  (* Name of the measurementw *)
    statuses : ServicesMeteoMeasurementStatuses;  (* Statuses of the state machine *)
  END_VAR
  VAR_IN_OUT
    {attribute 'OPC.UA.DA' := '0'}
    config : MeasurementConfig;  (* Reference to the config *)
  END_VAR

            statuses.enabledStatus( isEnabled := config.enabled );
statuses.healthStatus(
    superState := statuses.enabledStatus.enabled,
    isGood := NOT(invalidData OR (statuses.alarmStatus.hiHi OR statuses.alarmStatus.loLo)),
    hasWarning := statuses.alarmStatus.hi OR statuses.alarmStatus.lo);
statuses.alarmStatus(
    superState := statuses.enabledStatus.enabled,
    config := config.alarms,
    value := data.value);

          

{attribute 'TcRpcEnable' := '1'}
METHOD _log : BOOL
  VAR_INPUT
    name : STRING;  (* Name of this function block instance *)
  END_VAR
  VAR_IN_OUT
    buffer : LogBuffer;  (* Buffer to write all logging to *)
  END_VAR
  VAR
    subBuffer : LogBuffer;  (* Temporary buffer to write logging by parts (sub-statemachines) to *)
  END_VAR
                  LOGGER(
    name := name,
    actualStatus := THIS^.actualStatus,
    previousStatus := THIS^.previousStatus,
    buffer := buffer,
    subBuffer := subBuffer,
    pHealthStatus := ADR(THIS^.statuses.healthStatus));

                
END_METHOD
END_FUNCTION_BLOCK

FUNCTION_BLOCK SM_ServicesMeteo
  VAR_INPUT
    {attribute 'OPC.UA.DA' := '1'}
    {attribute 'OPC.UA.DA.Access' := '1'}
    serialTimeout : BOOL;  (* Is the serial data not being received within time? *)
    {attribute 'OPC.UA.DA' := '1'}
    {attribute 'OPC.UA.DA.Access' := '1'}
    comError : BOOL;  (* Is there any problem with the COM port? *)
    {attribute 'OPC.UA.DA' := '1'}
    {attribute 'OPC.UA.DA.Access' := '1'}
    comErrorID : INT;  (* COM error id (see Beckhoff ComError_t) *)
    {attribute 'OPC.UA.DA' := '1'}
    {attribute 'OPC.UA.DA.Access' := '1'}
    comErrorDescription : STRING;  (* Description of the COM error id *)
    {attribute 'OPC.UA.DA' := '1'}
    {attribute 'OPC.UA.DA.Access' := '1'}
    windSpeedMinimum : ServicesMeteoMeasurement;  (* Wind speed minimum *)
    {attribute 'OPC.UA.DA' := '1'}
    {attribute 'OPC.UA.DA.Access' := '1'}
    windSpeedAverage : ServicesMeteoMeasurement;  (* Wind speed average *)
    {attribute 'OPC.UA.DA' := '1'}
    {attribute 'OPC.UA.DA.Access' := '1'}
    windSpeedMaximum : ServicesMeteoMeasurement;  (* Wind speed maximum *)
    {attribute 'OPC.UA.DA' := '1'}
    {attribute 'OPC.UA.DA.Access' := '1'}
    windDirectionMinimum : ServicesMeteoMeasurement;  (* Wind direction minimum *)
    {attribute 'OPC.UA.DA' := '1'}
    {attribute 'OPC.UA.DA.Access' := '1'}
    windDirectionAverage : ServicesMeteoMeasurement;  (* Wind direction average *)
    {attribute 'OPC.UA.DA' := '1'}
    {attribute 'OPC.UA.DA.Access' := '1'}
    windDirectionMaximum : ServicesMeteoMeasurement;  (* Wind direction maximum *)
    {attribute 'OPC.UA.DA' := '1'}
    {attribute 'OPC.UA.DA.Access' := '1'}
    airPressure : ServicesMeteoMeasurement;  (* Air pressure *)
    {attribute 'OPC.UA.DA' := '1'}
    {attribute 'OPC.UA.DA.Access' := '1'}
    airTemperature : ServicesMeteoMeasurement;  (* Air temperature *)
    {attribute 'OPC.UA.DA' := '1'}
    {attribute 'OPC.UA.DA.Access' := '1'}
    internalTemperature : ServicesMeteoMeasurement;  (* Internal temperature *)
    {attribute 'OPC.UA.DA' := '1'}
    {attribute 'OPC.UA.DA.Access' := '1'}
    relativeHumidity : ServicesMeteoMeasurement;  (* Relative humidity *)
    {attribute 'OPC.UA.DA' := '1'}
    {attribute 'OPC.UA.DA.Access' := '1'}
    rainAccumulation : ServicesMeteoMeasurement;  (* Rain accumulation *)
    {attribute 'OPC.UA.DA' := '1'}
    {attribute 'OPC.UA.DA.Access' := '1'}
    rainDuration : ServicesMeteoMeasurement;  (* Rain duration *)
    {attribute 'OPC.UA.DA' := '1'}
    {attribute 'OPC.UA.DA.Access' := '1'}
    rainIntensity : ServicesMeteoMeasurement;  (* Rain intensity *)
    {attribute 'OPC.UA.DA' := '1'}
    {attribute 'OPC.UA.DA.Access' := '1'}
    rainPeakIntensity : ServicesMeteoMeasurement;  (* Rain peak intensity *)
    {attribute 'OPC.UA.DA' := '1'}
    {attribute 'OPC.UA.DA.Access' := '1'}
    hailAccumulation : ServicesMeteoMeasurement;  (* Hail accumulation *)
    {attribute 'OPC.UA.DA' := '1'}
    {attribute 'OPC.UA.DA.Access' := '1'}
    hailDuration : ServicesMeteoMeasurement;  (* Hail duration *)
    {attribute 'OPC.UA.DA' := '1'}
    {attribute 'OPC.UA.DA.Access' := '1'}
    hailIntensity : ServicesMeteoMeasurement;  (* Hail intensity *)
    {attribute 'OPC.UA.DA' := '1'}
    {attribute 'OPC.UA.DA.Access' := '1'}
    hailPeakIntensity : ServicesMeteoMeasurement;  (* Hail peak intensity *)
    {attribute 'OPC.UA.DA' := '1'}
    {attribute 'OPC.UA.DA.Access' := '1'}
    heatingTemperature : ServicesMeteoMeasurement;  (* Heating temperature *)
    {attribute 'OPC.UA.DA' := '1'}
    {attribute 'OPC.UA.DA.Access' := '1'}
    heatingVoltage : ServicesMeteoMeasurement;  (* Heating voltage *)
    {attribute 'OPC.UA.DA' := '1'}
    {attribute 'OPC.UA.DA.Access' := '1'}
    supplyVoltage : ServicesMeteoMeasurement;  (* Supply voltage *)
    {attribute 'OPC.UA.DA' := '1'}
    {attribute 'OPC.UA.DA.Access' := '1'}
    referenceVoltage : ServicesMeteoMeasurement;  (* Reference voltage *)
    {attribute 'OPC.UA.DA' := '1'}
    {attribute 'OPC.UA.DA.Access' := '1'}
    durationOK : Duration;  (* Duration that the meteo is OK *)
    {attribute 'OPC.UA.DA' := '1'}
    {attribute 'OPC.UA.DA.Access' := '1'}
    dewpoint : Temperature;  (* Calculated dewpoint *)
    {attribute 'OPC.UA.DA' := '1'}
    {attribute 'OPC.UA.DA.Access' := '1'}
    wet : BOOL;  (* Wet if (rainIntensity+hailIntensity) > config.wetLimit *)
    {attribute 'OPC.UA.DA' := '1'}
    {attribute 'OPC.UA.DA.Access' := '1'}
    heating : BOOL;  (* Heating or not? *)
    {attribute 'OPC.UA.DA' := '1'}
    {attribute 'OPC.UA.DA.Access' := '1'}
    windDirectionMinimumString : STRING;  (* Average direction of the wind as a string *)
    {attribute 'OPC.UA.DA' := '1'}
    {attribute 'OPC.UA.DA.Access' := '1'}
    windDirectionAverageString : STRING;  (* Average direction of the wind as a string *)
    {attribute 'OPC.UA.DA' := '1'}
    {attribute 'OPC.UA.DA.Access' := '1'}
    windDirectionMaximumString : STRING;  (* Average direction of the wind as a string *)
  END_VAR
  VAR_OUTPUT
    {attribute 'OPC.UA.DA' := '1'}
    {attribute 'OPC.UA.DA.Access' := '1'}
    actualStatus : STRING;  (* Current status description *)
    previousStatus : STRING;  (* Previous status description *)
    statuses : ServicesMeteoStatuses;  (* Statuses of the state machine *)
    processes : ServicesMeteoProcesses;  (* Processes of the state machine *)
  END_VAR
  VAR_IN_OUT
    {attribute 'OPC.UA.DA' := '0'}
    config : ServicesMeteoConfig;  (* The config *)
  END_VAR

            windSpeedMinimum(
    id := ServicesMeteoId.WIND_SPEED_MINIMUM,
    config := config.windSpeedMinimum);
windSpeedAverage(
    id := ServicesMeteoId.WIND_SPEED_AVERAGE,
    config := config.windSpeedAverage);
windSpeedMaximum(
    id := ServicesMeteoId.WIND_SPEED_MAXIMUM,
    config := config.windSpeedMaximum);
windDirectionMinimum(
    id := ServicesMeteoId.WIND_DIRECTION_MINIMUM,
    config := config.windDirectionMinimum);
windDirectionAverage(
    id := ServicesMeteoId.WIND_DIRECTION_AVERAGE,
    config := config.windDirectionAverage);
windDirectionMaximum(
    id := ServicesMeteoId.WIND_DIRECTION_MAXIMUM,
    config := config.windDirectionMaximum);
airPressure(
    id := ServicesMeteoId.AIR_PRESSURE,
    config := config.airPressure);
airTemperature(
    id := ServicesMeteoId.AIR_TEMPERATURE,
    config := config.airTemperature);
internalTemperature(
    id := ServicesMeteoId.INTERNAL_TEMPERATURE,
    config := config.internalTemperature);
relativeHumidity(
    id := ServicesMeteoId.RELATIVE_HUMIDITY,
    config := config.relativeHumidity);
rainAccumulation(
    id := ServicesMeteoId.RAIN_ACCUMULATION,
    config := config.rainAccumulation);
rainDuration(
    id := ServicesMeteoId.RAIN_DURATION,
    config := config.rainDuration);
rainIntensity(
    id := ServicesMeteoId.RAIN_INTENSITY,
    config := config.rainIntensity);
rainPeakIntensity(
    id := ServicesMeteoId.RAIN_PEAK_INTENSITY,
    config := config.rainPeakIntensity);
hailAccumulation(
    id := ServicesMeteoId.HAIL_ACCUMULATION,
    config := config.hailAccumulation);
hailDuration(
    id := ServicesMeteoId.HAIL_DURATION,
    config := config.hailDuration);
hailIntensity(
    id := ServicesMeteoId.HAIL_INTENSITY,
    config := config.hailIntensity);
hailPeakIntensity(
    id := ServicesMeteoId.HAIL_PEAK_INTENSITY,
    config := config.hailPeakIntensity);
heatingTemperature(
    id := ServicesMeteoId.HEATING_TEMPERATURE,
    config := config.heatingTemperature);
heatingVoltage(
    id := ServicesMeteoId.HEATING_VOLTAGE,
    config := config.heatingVoltage);
supplyVoltage(
    id := ServicesMeteoId.SUPPLY_VOLTAGE,
    config := config.supplyVoltage);
referenceVoltage(
    id := ServicesMeteoId.REFERENCE_VOLTAGE,
    config := config.referenceVoltage);
statuses.meteoHealthStatus(
    superState := statuses.healthStatus.good,
    isGood := (windSpeedMinimum.statuses.healthStatus.isGood OR windSpeedMinimum.statuses.enabledStatus.disabled) AND ((windSpeedAverage.statuses.healthStatus.isGood OR windSpeedAverage.statuses.enabledStatus.disabled) AND ((windSpeedMaximum.statuses.healthStatus.isGood OR windSpeedMaximum.statuses.enabledStatus.disabled) AND ((windDirectionMinimum.statuses.healthStatus.isGood OR windDirectionMinimum.statuses.enabledStatus.disabled) AND ((windDirectionAverage.statuses.healthStatus.isGood OR windDirectionAverage.statuses.enabledStatus.disabled) AND ((windDirectionMaximum.statuses.healthStatus.isGood OR windDirectionMaximum.statuses.enabledStatus.disabled) AND ((airPressure.statuses.healthStatus.isGood OR airPressure.statuses.enabledStatus.disabled) AND ((airTemperature.statuses.healthStatus.isGood OR airTemperature.statuses.enabledStatus.disabled) AND ((internalTemperature.statuses.healthStatus.isGood OR internalTemperature.statuses.enabledStatus.disabled) AND ((relativeHumidity.statuses.healthStatus.isGood OR relativeHumidity.statuses.enabledStatus.disabled) AND ((rainAccumulation.statuses.healthStatus.isGood OR rainAccumulation.statuses.enabledStatus.disabled) AND ((rainDuration.statuses.healthStatus.isGood OR rainDuration.statuses.enabledStatus.disabled) AND ((rainIntensity.statuses.healthStatus.isGood OR rainIntensity.statuses.enabledStatus.disabled) AND ((rainPeakIntensity.statuses.healthStatus.isGood OR rainPeakIntensity.statuses.enabledStatus.disabled) AND ((hailAccumulation.statuses.healthStatus.isGood OR hailAccumulation.statuses.enabledStatus.disabled) AND ((hailDuration.statuses.healthStatus.isGood OR hailDuration.statuses.enabledStatus.disabled) AND ((hailIntensity.statuses.healthStatus.isGood OR hailIntensity.statuses.enabledStatus.disabled) AND ((hailPeakIntensity.statuses.healthStatus.isGood OR hailPeakIntensity.statuses.enabledStatus.disabled) AND ((heatingTemperature.statuses.healthStatus.isGood OR heatingTemperature.statuses.enabledStatus.disabled) AND ((heatingVoltage.statuses.healthStatus.isGood OR heatingVoltage.statuses.enabledStatus.disabled) AND ((supplyVoltage.statuses.healthStatus.isGood OR supplyVoltage.statuses.enabledStatus.disabled) AND (referenceVoltage.statuses.healthStatus.isGood OR referenceVoltage.statuses.enabledStatus.disabled))))))))))))))))))))),
    hasWarning := windSpeedMinimum.statuses.healthStatus.hasWarning OR (windSpeedAverage.statuses.healthStatus.hasWarning OR (windSpeedMaximum.statuses.healthStatus.hasWarning OR (windDirectionMinimum.statuses.healthStatus.hasWarning OR (windDirectionAverage.statuses.healthStatus.hasWarning OR (windDirectionMaximum.statuses.healthStatus.hasWarning OR (airPressure.statuses.healthStatus.hasWarning OR (airTemperature.statuses.healthStatus.hasWarning OR (internalTemperature.statuses.healthStatus.hasWarning OR (relativeHumidity.statuses.healthStatus.hasWarning OR (rainAccumulation.statuses.healthStatus.hasWarning OR (rainDuration.statuses.healthStatus.hasWarning OR (rainIntensity.statuses.healthStatus.hasWarning OR (rainPeakIntensity.statuses.healthStatus.hasWarning OR (hailAccumulation.statuses.healthStatus.hasWarning OR (hailDuration.statuses.healthStatus.hasWarning OR (hailIntensity.statuses.healthStatus.hasWarning OR (hailPeakIntensity.statuses.healthStatus.hasWarning OR (heatingTemperature.statuses.healthStatus.hasWarning OR (heatingVoltage.statuses.healthStatus.hasWarning OR (supplyVoltage.statuses.healthStatus.hasWarning OR referenceVoltage.statuses.healthStatus.hasWarning)))))))))))))))))))));
statuses.healthStatus( isGood := NOT(serialTimeout OR comError) );

          

{attribute 'TcRpcEnable' := '1'}
METHOD _log : BOOL
  VAR_INPUT
    name : STRING;  (* Name of this function block instance *)
  END_VAR
  VAR_IN_OUT
    buffer : LogBuffer;  (* Buffer to write all logging to *)
  END_VAR
  VAR
    subBuffer : LogBuffer;  (* Temporary buffer to write logging by parts (sub-statemachines) to *)
  END_VAR
                  LOGGER(
    name := name,
    actualStatus := THIS^.actualStatus,
    previousStatus := THIS^.previousStatus,
    buffer := buffer,
    subBuffer := subBuffer,
    pHealthStatus := ADR(THIS^.statuses.healthStatus));

                
END_METHOD
END_FUNCTION_BLOCK

FUNCTION_BLOCK SM_ServicesWestController
  VAR_INPUT
    {attribute 'OPC.UA.DA' := '1'}
    {attribute 'OPC.UA.DA.Access' := '1'}
    isEnabled : BOOL;  (* Are the processes enabled? *)
    {attribute 'OPC.UA.DA' := '1'}
    {attribute 'OPC.UA.DA.Access' := '1'}
    manualControl : BOOL;  (* Controller switched to manualControl *)
    {attribute 'OPC.UA.DA' := '1'}
    {attribute 'OPC.UA.DA.Access' := '1'}
    unit : Units;
    {attribute 'OPC.UA.DA' := '1'}
    {attribute 'OPC.UA.DA.Access' := '1'}
    setpoint : QuantityValue;  (* The current setpoint *)
    {attribute 'OPC.UA.DA' := '1'}
    {attribute 'OPC.UA.DA.Access' := '1'}
    defaultSetpoint : QuantityValue;  (* The default setpoint *)
    {attribute 'OPC.UA.DA' := '1'}
    {attribute 'OPC.UA.DA.Access' := '1'}
    minSetpoint : QuantityValue;  (* The minimun setpoint *)
    {attribute 'OPC.UA.DA' := '1'}
    {attribute 'OPC.UA.DA.Access' := '1'}
    maxSetpoint : QuantityValue;  (* The maximal setpoint *)
    {attribute 'OPC.UA.DA' := '1'}
    {attribute 'OPC.UA.DA.Access' := '1'}
    offset : QuantityValue;  (* Offset internally added to Process Value *)
    {attribute 'OPC.UA.DA' := '1'}
    {attribute 'OPC.UA.DA.Access' := '1'}
    differentialOnOff : QuantityValue;  (* Differential band for On/Off *)
    {attribute 'OPC.UA.DA' := '1'}
    {attribute 'OPC.UA.DA.Access' := '1'}
    alarmValue : QuantityValue;  (* Alarm value from setpoint *)
    {attribute 'OPC.UA.DA' := '1'}
    {attribute 'OPC.UA.DA.Access' := '1'}
    inputFilter : QuantityValue;  (* Input input filter time constant *)
    {attribute 'OPC.UA.DA' := '1'}
    {attribute 'OPC.UA.DA.Access' := '1'}
    cycleTime : QuantityValue;  (* Cycle time for control loop *)
    {attribute 'OPC.UA.DA' := '1'}
    {attribute 'OPC.UA.DA.Access' := '1'}
    proportionalBand : QuantityValue;  (* Proportional band constant *)
    {attribute 'OPC.UA.DA' := '1'}
    {attribute 'OPC.UA.DA.Access' := '1'}
    resetTime : QuantityValue;  (* Integral time constant *)
    {attribute 'OPC.UA.DA' := '1'}
    {attribute 'OPC.UA.DA.Access' := '1'}
    rate : QuantityValue;  (* Derivative time constant *)
    {attribute 'OPC.UA.DA' := '1'}
    {attribute 'OPC.UA.DA.Access' := '1'}
    outputPower : QuantityValue;  (* The Output power in percentage *)
  END_VAR
  VAR_OUTPUT
    {attribute 'OPC.UA.DA' := '1'}
    {attribute 'OPC.UA.DA.Access' := '1'}
    actualStatus : STRING;  (* Current status description *)
    previousStatus : STRING;  (* Previous status description *)
    {attribute 'OPC.UA.DA' := '1'}
    {attribute 'OPC.UA.DA.Access' := '1'}
    invalidData : BOOL;  (* True if there is invalid data *)
    {attribute 'OPC.UA.DA' := '1'}
    {attribute 'OPC.UA.DA.Access' := '1'}
    processValue : QuantityValue;  (* The Process value *)
    {attribute 'OPC.UA.DA' := '1'}
    {attribute 'OPC.UA.DA.Access' := '1'}
    alarmActivated : BOOL;  (* True if controller alarm is activated *)
    statuses : ServicesWestControllerStatuses;  (* Statuses of the state machine *)
    processes : ServicesWestControllerProcesses;  (* Processes of the state machine *)
  END_VAR
  VAR_IN_OUT
    {attribute 'OPC.UA.DA' := '0'}
    config : ServicesWestControllerConfig;  (* A small config only for a single WEST controller *)
    {attribute 'OPC.UA.DA' := '0'}
    bus : ModbusRTUBus;  (* The shared Modbus RTU bus *)
  END_VAR

            statuses.healthStatus(
    superState := config.measurement.enabled,
    isGood := NOT(invalidData OR (statuses.alarmStatus.hiHi OR statuses.alarmStatus.loLo)),
    hasWarning := statuses.alarmStatus.hi OR statuses.alarmStatus.lo);
statuses.alarmStatus(
    superState := config.measurement.enabled,
    config := config.measurement.alarms,
    value := processValue.value);
processes.updateProcessVariables( isEnabled := isEnabled );
processes.updateConfigVariables( isEnabled := isEnabled );
processes.writeSetpoint( isEnabled := isEnabled );
processes.writeOffset( isEnabled := isEnabled );
processes.writeProportinalBand( isEnabled := isEnabled );
processes.writeResetTime( isEnabled := isEnabled );
processes.writeRate( isEnabled := isEnabled );
processes.switchToManual( isEnabled := isEnabled );
processes.switchToAuto( isEnabled := isEnabled );
processes.writeOutputPower( isEnabled := isEnabled );
processes.writeConfigToController( isEnabled := isEnabled );

          

{attribute 'TcRpcEnable' := '1'}
METHOD updateProcessVariables : RequestResults
                  updateProcessVariables := THIS^.processes.updateProcessVariables.request();

                
END_METHOD

{attribute 'TcRpcEnable' := '1'}
METHOD updateConfigVariables : RequestResults
                  updateConfigVariables := THIS^.processes.updateConfigVariables.request();

                
END_METHOD

{attribute 'TcRpcEnable' := '1'}
METHOD writeSetpoint : RequestResults
  VAR_INPUT
    setpoint : LREAL;
  END_VAR
                  writeSetpoint := THIS^.processes.writeSetpoint.request( setpoint := setpoint );

                
END_METHOD

{attribute 'TcRpcEnable' := '1'}
METHOD writeOffset : RequestResults
  VAR_INPUT
    parameter : LREAL;
  END_VAR
                  writeOffset := THIS^.processes.writeOffset.request( parameter := parameter );

                
END_METHOD

{attribute 'TcRpcEnable' := '1'}
METHOD writeProportinalBand : RequestResults
  VAR_INPUT
    parameter : LREAL;
  END_VAR
                  writeProportinalBand := THIS^.processes.writeProportinalBand.request( parameter := parameter );

                
END_METHOD

{attribute 'TcRpcEnable' := '1'}
METHOD writeResetTime : RequestResults
  VAR_INPUT
    parameter : LREAL;
  END_VAR
                  writeResetTime := THIS^.processes.writeResetTime.request( parameter := parameter );

                
END_METHOD

{attribute 'TcRpcEnable' := '1'}
METHOD writeRate : RequestResults
  VAR_INPUT
    parameter : LREAL;
  END_VAR
                  writeRate := THIS^.processes.writeRate.request( parameter := parameter );

                
END_METHOD

{attribute 'TcRpcEnable' := '1'}
METHOD switchToManual : RequestResults
                  switchToManual := THIS^.processes.switchToManual.request();

                
END_METHOD

{attribute 'TcRpcEnable' := '1'}
METHOD switchToAuto : RequestResults
                  switchToAuto := THIS^.processes.switchToAuto.request();

                
END_METHOD

{attribute 'TcRpcEnable' := '1'}
METHOD writeOutputPower : RequestResults
  VAR_INPUT
    parameter : LREAL;
  END_VAR
                  writeOutputPower := THIS^.processes.writeOutputPower.request( parameter := parameter );

                
END_METHOD

{attribute 'TcRpcEnable' := '1'}
METHOD writeConfigToController : RequestResults
                  writeConfigToController := THIS^.processes.writeConfigToController.request();

                
END_METHOD

{attribute 'TcRpcEnable' := '1'}
METHOD _log : BOOL
  VAR_INPUT
    name : STRING;  (* Name of this function block instance *)
  END_VAR
  VAR_IN_OUT
    buffer : LogBuffer;  (* Buffer to write all logging to *)
  END_VAR
  VAR
    subBuffer : LogBuffer;  (* Temporary buffer to write logging by parts (sub-statemachines) to *)
  END_VAR
                  THIS^.processes.updateProcessVariables._log(
    name := 'processes.updateProcessVariables',
    buffer := subBuffer);
THIS^.processes.updateConfigVariables._log(
    name := 'processes.updateConfigVariables',
    buffer := subBuffer);
THIS^.processes.writeSetpoint._log(
    name := 'processes.writeSetpoint',
    buffer := subBuffer);
THIS^.processes.writeOffset._log(
    name := 'processes.writeOffset',
    buffer := subBuffer);
THIS^.processes.writeProportinalBand._log(
    name := 'processes.writeProportinalBand',
    buffer := subBuffer);
THIS^.processes.writeResetTime._log(
    name := 'processes.writeResetTime',
    buffer := subBuffer);
THIS^.processes.writeRate._log(
    name := 'processes.writeRate',
    buffer := subBuffer);
THIS^.processes.switchToManual._log(
    name := 'processes.switchToManual',
    buffer := subBuffer);
THIS^.processes.switchToAuto._log(
    name := 'processes.switchToAuto',
    buffer := subBuffer);
THIS^.processes.writeOutputPower._log(
    name := 'processes.writeOutputPower',
    buffer := subBuffer);
THIS^.processes.writeConfigToController._log(
    name := 'processes.writeConfigToController',
    buffer := subBuffer);
LOGGER(
    name := name,
    actualStatus := THIS^.actualStatus,
    previousStatus := THIS^.previousStatus,
    buffer := buffer,
    subBuffer := subBuffer,
    pHealthStatus := ADR(THIS^.statuses.healthStatus));

                
END_METHOD
END_FUNCTION_BLOCK

FUNCTION_BLOCK SM_ServicesWest
  VAR_OUTPUT
    {attribute 'OPC.UA.DA' := '1'}
    {attribute 'OPC.UA.DA.Access' := '1'}
    actualStatus : STRING;  (* Current status description *)
    previousStatus : STRING;  (* Previous status description *)
    statuses : ServicesWestStatuses;  (* Statuses of the state machine *)
    parts : ServicesWestParts;  (* Parts of the state machine *)
    processes : ServicesWestProcesses;  (* Processes of the state machine *)
  END_VAR
  VAR_IN_OUT
    {attribute 'OPC.UA.DA' := '0'}
    operatorStatus : OperatorStatus;  (* Shared operator status *)
    {attribute 'OPC.UA.DA' := '0'}
    config : ServicesWestConfig;  (* The config *)
    {attribute 'OPC.UA.DA' := '0'}
    airTemperature : ServicesMeteoMeasurement;  (* Air temperature *)
    {attribute 'OPC.UA.DA' := '0'}
    domeApertureStatus : ApertureStatus;  (* Is the dome open or closed? *)
  END_VAR

            parts.bus( isEnabled := operatorStatus.tech AND statuses.operatingStatus.manual );
parts.domeTemperature(
    isEnabled := parts.bus.isEnabled,
    unit := Units.DEGREES_CELSIUS,
    config := config.domeTemperature,
    bus := parts.bus);
parts.firstFloorTemperature(
    isEnabled := parts.bus.isEnabled,
    unit := Units.DEGREES_CELSIUS,
    config := config.firstFloorTemperature,
    bus := parts.bus);
parts.pumpsRoomTemperature(
    isEnabled := parts.bus.isEnabled,
    unit := Units.DEGREES_CELSIUS,
    config := config.pumpsRoomTemperature,
    bus := parts.bus);
parts.oilHeatExchangerTemperature(
    isEnabled := parts.bus.isEnabled,
    unit := Units.DEGREES_CELSIUS,
    config := config.oilHeatExchangerTemperature,
    bus := parts.bus);
parts.serversRoomTemperature(
    isEnabled := parts.bus.isEnabled,
    unit := Units.DEGREES_CELSIUS,
    config := config.serversRoomTemperature,
    bus := parts.bus);
statuses.healthStatus(
    isGood := parts.domeTemperature.statuses.healthStatus.isGood AND (parts.firstFloorTemperature.statuses.healthStatus.isGood AND (parts.pumpsRoomTemperature.statuses.healthStatus.isGood AND (parts.oilHeatExchangerTemperature.statuses.healthStatus.isGood AND parts.serversRoomTemperature.statuses.healthStatus.isGood))),
    hasWarning := parts.domeTemperature.statuses.healthStatus.hasWarning OR (parts.firstFloorTemperature.statuses.healthStatus.hasWarning OR (parts.pumpsRoomTemperature.statuses.healthStatus.hasWarning OR (parts.oilHeatExchangerTemperature.statuses.healthStatus.hasWarning OR parts.serversRoomTemperature.statuses.healthStatus.hasWarning))));
statuses.operatingStatus();
processes.changeOperatingState( isEnabled := operatorStatus.tech );

          

{attribute 'TcRpcEnable' := '1'}
METHOD changeOperatingState : RequestResults
  VAR_INPUT
    state : OperatingStates;
  END_VAR
                  changeOperatingState := THIS^.processes.changeOperatingState.request( state := state );

                
END_METHOD

{attribute 'TcRpcEnable' := '1'}
METHOD _log : BOOL
  VAR_INPUT
    name : STRING;  (* Name of this function block instance *)
  END_VAR
  VAR_IN_OUT
    buffer : LogBuffer;  (* Buffer to write all logging to *)
  END_VAR
  VAR
    subBuffer : LogBuffer;  (* Temporary buffer to write logging by parts (sub-statemachines) to *)
  END_VAR
                  THIS^.parts.bus._log(
    name := 'bus',
    buffer := subBuffer);
THIS^.parts.domeTemperature._log(
    name := 'domeTemperature',
    buffer := subBuffer);
THIS^.parts.firstFloorTemperature._log(
    name := 'firstFloorTemperature',
    buffer := subBuffer);
THIS^.parts.pumpsRoomTemperature._log(
    name := 'pumpsRoomTemperature',
    buffer := subBuffer);
THIS^.parts.oilHeatExchangerTemperature._log(
    name := 'oilHeatExchangerTemperature',
    buffer := subBuffer);
THIS^.parts.serversRoomTemperature._log(
    name := 'serversRoomTemperature',
    buffer := subBuffer);
THIS^.processes.changeOperatingState._log(
    name := 'processes.changeOperatingState',
    buffer := subBuffer);
LOGGER(
    name := name,
    actualStatus := THIS^.actualStatus,
    previousStatus := THIS^.previousStatus,
    buffer := buffer,
    subBuffer := subBuffer,
    pHealthStatus := ADR(THIS^.statuses.healthStatus));

                
END_METHOD
END_FUNCTION_BLOCK

FUNCTION_BLOCK SM_ServicesChillerController
  VAR_INPUT
    {attribute 'OPC.UA.DA' := '1'}
    {attribute 'OPC.UA.DA.Access' := '1'}
    isEnabled : BOOL;  (* Are the processes enabled? *)
    {attribute 'OPC.UA.DA' := '1'}
    {attribute 'OPC.UA.DA.Access' := '1'}
    chillerOn : BOOL;  (* The unit status, TRUE = Chiller is ON *)
    {attribute 'OPC.UA.DA' := '1'}
    {attribute 'OPC.UA.DA.Access' := '1'}
    resetAlarmRegisters : BOOL;  (* Flag to reset all active alarms *)
    {attribute 'OPC.UA.DA' := '1'}
    {attribute 'OPC.UA.DA.Access' := '1'}
    setpoint : QuantityValue;  (* The setpoint *)
    {attribute 'OPC.UA.DA' := '1'}
    {attribute 'OPC.UA.DA.Access' := '1'}
    minSetpoint : QuantityValue;  (* The minimun setpoint *)
    {attribute 'OPC.UA.DA' := '1'}
    {attribute 'OPC.UA.DA.Access' := '1'}
    maxSetpoint : QuantityValue;  (* The maximal setpoint *)
    {attribute 'OPC.UA.DA' := '1'}
    {attribute 'OPC.UA.DA.Access' := '1'}
    trippingBand : QuantityValue;  (* The tripping band *)
    {attribute 'OPC.UA.DA' := '1'}
    {attribute 'OPC.UA.DA.Access' := '1'}
    unitStatus : QuantityValue;  (* The unit status *)
    {attribute 'OPC.UA.DA' := '1'}
    {attribute 'OPC.UA.DA.Access' := '1'}
    unitResetRegister : QuantityValue;  (* The unit reset register *)
    {attribute 'OPC.UA.DA' := '1'}
    {attribute 'OPC.UA.DA.Access' := '1'}
    hoursCompressor1 : QuantityValue;  (* Operation hours of compressor 1 *)
    {attribute 'OPC.UA.DA' := '1'}
    {attribute 'OPC.UA.DA.Access' := '1'}
    hoursCompressor2 : QuantityValue;  (* Operation hours of compressor 2 *)
    {attribute 'OPC.UA.DA' := '1'}
    {attribute 'OPC.UA.DA.Access' := '1'}
    hoursCompressor3 : QuantityValue;  (* Operation hours of compressor 3 *)
    {attribute 'OPC.UA.DA' := '1'}
    {attribute 'OPC.UA.DA.Access' := '1'}
    hoursCompressor4 : QuantityValue;  (* Operation hours of compressor 4 *)
    {attribute 'OPC.UA.DA' := '1'}
    {attribute 'OPC.UA.DA.Access' := '1'}
    hoursPump : QuantityValue;  (* Operation hours of water pump *)
  END_VAR
  VAR_OUTPUT
    {attribute 'OPC.UA.DA' := '1'}
    {attribute 'OPC.UA.DA.Access' := '1'}
    actualStatus : STRING;  (* Current status description *)
    previousStatus : STRING;  (* Previous status description *)
    {attribute 'OPC.UA.DA' := '1'}
    {attribute 'OPC.UA.DA.Access' := '1'}
    invalidData : BOOL;  (* True if there is invalid data *)
    {attribute 'OPC.UA.DA' := '1'}
    {attribute 'OPC.UA.DA.Access' := '1'}
    waterTankTemperature : QuantityValue;  (* Water tank temperature *)
    {attribute 'OPC.UA.DA' := '1'}
    {attribute 'OPC.UA.DA.Access' := '1'}
    highPressureCircuit1 : QuantityValue;  (* High pressure of circuit 1 *)
    {attribute 'OPC.UA.DA' := '1'}
    {attribute 'OPC.UA.DA.Access' := '1'}
    highPressureCircuit2 : QuantityValue;  (* High pressure of circuit 2 *)
    {attribute 'OPC.UA.DA' := '1'}
    {attribute 'OPC.UA.DA.Access' := '1'}
    chillerCurrentInput : QuantityValue;  (* Chiller current input *)
    {attribute 'OPC.UA.DA' := '1'}
    {attribute 'OPC.UA.DA.Access' := '1'}
    waterPumpCurrentInput : QuantityValue;  (* Water pump current input *)
    {attribute 'OPC.UA.DA' := '1'}
    {attribute 'OPC.UA.DA.Access' := '1'}
    evaporatorOutTemp1 : QuantityValue;  (* Evaporator out temperature 1 *)
    {attribute 'OPC.UA.DA' := '1'}
    {attribute 'OPC.UA.DA.Access' := '1'}
    evaporatorOutTemp2 : QuantityValue;  (* EvaporwaterTankTemperatureMeasurementator out temperature 2 *)
    {attribute 'OPC.UA.DA' := '1'}
    {attribute 'OPC.UA.DA.Access' := '1'}
    ambientTemperature : QuantityValue;  (* Ambient temperature *)
    {attribute 'OPC.UA.DA' := '1'}
    {attribute 'OPC.UA.DA.Access' := '1'}
    waterPumpChassisTemp : QuantityValue;  (* Water Pump chassis temperature *)
    {attribute 'OPC.UA.DA' := '1'}
    {attribute 'OPC.UA.DA.Access' := '1'}
    flowSwitchStatus : BOOL;  (* Flow switch status. Digital Input Status 1 *)
    {attribute 'OPC.UA.DA' := '1'}
    {attribute 'OPC.UA.DA.Access' := '1'}
    digitalInputStatus2 : BOOL;  (* Digital input status 2 *)
    {attribute 'OPC.UA.DA' := '1'}
    {attribute 'OPC.UA.DA.Access' := '1'}
    digitalInputStatus3 : BOOL;  (* Digital input status 3 *)
    {attribute 'OPC.UA.DA' := '1'}
    {attribute 'OPC.UA.DA.Access' := '1'}
    digitalInputStatus4 : BOOL;  (* Digital input status 4 *)
    {attribute 'OPC.UA.DA' := '1'}
    {attribute 'OPC.UA.DA.Access' := '1'}
    alarmRelayOutput : BOOL;  (* Alarm output relay output status 1 *)
    {attribute 'OPC.UA.DA' := '1'}
    {attribute 'OPC.UA.DA.Access' := '1'}
    waterPumpRelayOutput : BOOL;  (* Water pump output relay output status 1 *)
    {attribute 'OPC.UA.DA' := '1'}
    {attribute 'OPC.UA.DA.Access' := '1'}
    relayOutputStatus2 : BOOL;  (* Relay output status 2 *)
    {attribute 'OPC.UA.DA' := '1'}
    {attribute 'OPC.UA.DA.Access' := '1'}
    relayOutputStatus3 : BOOL;  (* Relay output status 3 *)
    {attribute 'OPC.UA.DA' := '1'}
    {attribute 'OPC.UA.DA.Access' := '1'}
    compressorStatus1 : BOOL;  (* Compressor 1 status. ON/OFF *)
    {attribute 'OPC.UA.DA' := '1'}
    {attribute 'OPC.UA.DA.Access' := '1'}
    compressorStatus2 : BOOL;  (* Compressor 2 status. ON/OFF *)
    {attribute 'OPC.UA.DA' := '1'}
    {attribute 'OPC.UA.DA.Access' := '1'}
    compressorStatus3 : BOOL;  (* Compressor 3 status. ON/OFF *)
    {attribute 'OPC.UA.DA' := '1'}
    {attribute 'OPC.UA.DA.Access' := '1'}
    compressorStatus4 : BOOL;  (* Compressor 4 status. ON/OFF *)
    {attribute 'OPC.UA.DA' := '1'}
    {attribute 'OPC.UA.DA.Access' := '1'}
    fanCondenser1Output : QuantityValue;  (* Fan condenser 1 analog output 1 *)
    {attribute 'OPC.UA.DA' := '1'}
    {attribute 'OPC.UA.DA.Access' := '1'}
    fanCondenser2Output : QuantityValue;  (* Fan condenser 2 analog output 2 *)
    {attribute 'OPC.UA.DA' := '1'}
    {attribute 'OPC.UA.DA.Access' := '1'}
    alarmStatus1 : QuantityValue;  (* Alarms bitwise register *)
    {attribute 'OPC.UA.DA' := '1'}
    {attribute 'OPC.UA.DA.Access' := '1'}
    alarmStatus2 : QuantityValue;  (* Alarms bitwise register *)
    {attribute 'OPC.UA.DA' := '1'}
    {attribute 'OPC.UA.DA.Access' := '1'}
    alarmStatus3 : QuantityValue;  (* Alarms bitwise register *)
    {attribute 'OPC.UA.DA' := '1'}
    {attribute 'OPC.UA.DA.Access' := '1'}
    alarmStatus6 : QuantityValue;  (* Alarms bitwise register *)
    {attribute 'OPC.UA.DA' := '1'}
    {attribute 'OPC.UA.DA.Access' := '1'}
    alarmStatus7 : QuantityValue;  (* Alarms bitwise register *)
    {attribute 'OPC.UA.DA' := '1'}
    {attribute 'OPC.UA.DA.Access' := '1'}
    alarmStatus10 : QuantityValue;  (* Alarms bitwise register *)
    {attribute 'OPC.UA.DA' := '1'}
    {attribute 'OPC.UA.DA.Access' := '1'}
    alarmStatus11 : QuantityValue;  (* Alarms bitwise register *)
    {attribute 'OPC.UA.DA' := '1'}
    {attribute 'OPC.UA.DA.Access' := '1'}
    alarmOilCompressor1 : QuantityValue;  (* Alarms per hour. Oil Compressor 1 *)
    {attribute 'OPC.UA.DA' := '1'}
    {attribute 'OPC.UA.DA.Access' := '1'}
    alarmOilCompressor2 : QuantityValue;  (* Alarms per hour. Oil Compressor 2 *)
    {attribute 'OPC.UA.DA' := '1'}
    {attribute 'OPC.UA.DA.Access' := '1'}
    alarmOilCompressor3 : QuantityValue;  (* Alarms per hour. Oil Compressor 3 *)
    {attribute 'OPC.UA.DA' := '1'}
    {attribute 'OPC.UA.DA.Access' := '1'}
    alarmOilCompressor4 : QuantityValue;  (* Alarms per hour. Oil Compressedor 4 *)
    {attribute 'OPC.UA.DA' := '1'}
    {attribute 'OPC.UA.DA.Access' := '1'}
    alarmFanOverload : QuantityValue;  (* Alarms per hour. Fan overload *)
    {attribute 'OPC.UA.DA' := '1'}
    {attribute 'OPC.UA.DA.Access' := '1'}
    alarmColdSideFlowSwitch : QuantityValue;  (* Alarms per hour. ColdSideFlowSwitch *)
    {attribute 'OPC.UA.DA' := '1'}
    {attribute 'OPC.UA.DA.Access' := '1'}
    alarmHotSideFlowSwitch : QuantityValue;  (* Alarms per hour. HotSideFlowSwitch *)
    {attribute 'OPC.UA.DA' := '1'}
    {attribute 'OPC.UA.DA.Access' := '1'}
    alarmCirc1LowTempPressDI : QuantityValue;  (* Alarms per hour. Circ1LowTempPressDI *)
    {attribute 'OPC.UA.DA' := '1'}
    {attribute 'OPC.UA.DA.Access' := '1'}
    alarmCirc2LowTempPressDI : QuantityValue;  (* Alarms per hour. Circ1LowTempPressPB *)
    {attribute 'OPC.UA.DA' := '1'}
    {attribute 'OPC.UA.DA.Access' := '1'}
    alarmCirc1LowTempPressPB : QuantityValue;  (* Alarms per hour. Circ1LowTempPressPB *)
    {attribute 'OPC.UA.DA' := '1'}
    {attribute 'OPC.UA.DA.Access' := '1'}
    alarmCirc2LowTempPressPB : QuantityValue;  (* Alarms per hour. Circ2LowTempPressPB *)
    statuses : ServicesChillerControllerStatuses;  (* Statuses of the state machine *)
    processes : ServicesChillerControllerProcesses;  (* Processes of the state machine *)
  END_VAR
  VAR_IN_OUT
    {attribute 'OPC.UA.DA' := '0'}
    config : ServicesChillerControllerConfig;  (* A small config only for Chiller controller *)
    {attribute 'OPC.UA.DA' := '0'}
    bus : ModbusRTUBus;  (* The shared Modbus RTU bus *)
  END_VAR

            statuses.healthStatus(
    superState := config.waterTankTemperatureMeasurement.enabled AND config.waterPumpSupervisorMeasurement.enabled,
    isGood := NOT(invalidData OR (alarmRelayOutput OR (statuses.alarmStatusWatertemperature.hiHi OR (statuses.alarmStatusWatertemperature.loLo OR (statuses.alarmStatusWaterPumpSupervisor.hiHi OR statuses.alarmStatusWaterPumpSupervisor.loLo))))),
    hasWarning := (NOT(chillerOn)) OR (flowSwitchStatus OR (statuses.alarmStatusWatertemperature.hi OR (statuses.alarmStatusWatertemperature.lo OR (statuses.alarmStatusWaterPumpSupervisor.hi OR statuses.alarmStatusWaterPumpSupervisor.lo)))));
statuses.alarmStatusWatertemperature(
    superState := config.waterTankTemperatureMeasurement.enabled,
    config := config.waterTankTemperatureMeasurement.alarms,
    value := waterTankTemperature.value);
statuses.alarmStatusWaterPumpSupervisor(
    superState := config.waterPumpSupervisorMeasurement.enabled,
    config := config.waterPumpSupervisorMeasurement.alarms,
    value := waterPumpCurrentInput.value);
processes.updateConfigVariables( isEnabled := isEnabled );
processes.updateMeasureVariables( isEnabled := isEnabled );
processes.updateAlarmRegisters( isEnabled := isEnabled );
processes.writeSetpoint( isEnabled := isEnabled );
processes.switchChillerON( isEnabled := isEnabled );
processes.switchChillerOFF( isEnabled := isEnabled );
processes.resetUnitController();
processes.resetAlarms( isEnabled := isEnabled );

          

{attribute 'TcRpcEnable' := '1'}
METHOD updateConfigVariables : RequestResults
                  updateConfigVariables := THIS^.processes.updateConfigVariables.request();

                
END_METHOD

{attribute 'TcRpcEnable' := '1'}
METHOD updateMeasureVariables : RequestResults
                  updateMeasureVariables := THIS^.processes.updateMeasureVariables.request();

                
END_METHOD

{attribute 'TcRpcEnable' := '1'}
METHOD updateAlarmRegisters : RequestResults
                  updateAlarmRegisters := THIS^.processes.updateAlarmRegisters.request();

                
END_METHOD

{attribute 'TcRpcEnable' := '1'}
METHOD writeSetpoint : RequestResults
  VAR_INPUT
    setpoint : LREAL;
  END_VAR
                  writeSetpoint := THIS^.processes.writeSetpoint.request( setpoint := setpoint );

                
END_METHOD

{attribute 'TcRpcEnable' := '1'}
METHOD switchChillerON : RequestResults
                  switchChillerON := THIS^.processes.switchChillerON.request();

                
END_METHOD

{attribute 'TcRpcEnable' := '1'}
METHOD switchChillerOFF : RequestResults
                  switchChillerOFF := THIS^.processes.switchChillerOFF.request();

                
END_METHOD

{attribute 'TcRpcEnable' := '1'}
METHOD resetUnitController : RequestResults
                  resetUnitController := THIS^.processes.resetUnitController.request();

                
END_METHOD

{attribute 'TcRpcEnable' := '1'}
METHOD resetAlarms : RequestResults
                  resetAlarms := THIS^.processes.resetAlarms.request();

                
END_METHOD

{attribute 'TcRpcEnable' := '1'}
METHOD _log : BOOL
  VAR_INPUT
    name : STRING;  (* Name of this function block instance *)
  END_VAR
  VAR_IN_OUT
    buffer : LogBuffer;  (* Buffer to write all logging to *)
  END_VAR
  VAR
    subBuffer : LogBuffer;  (* Temporary buffer to write logging by parts (sub-statemachines) to *)
  END_VAR
                  THIS^.processes.updateConfigVariables._log(
    name := 'processes.updateConfigVariables',
    buffer := subBuffer);
THIS^.processes.updateMeasureVariables._log(
    name := 'processes.updateMeasureVariables',
    buffer := subBuffer);
THIS^.processes.updateAlarmRegisters._log(
    name := 'processes.updateAlarmRegisters',
    buffer := subBuffer);
THIS^.processes.writeSetpoint._log(
    name := 'processes.writeSetpoint',
    buffer := subBuffer);
THIS^.processes.switchChillerON._log(
    name := 'processes.switchChillerON',
    buffer := subBuffer);
THIS^.processes.switchChillerOFF._log(
    name := 'processes.switchChillerOFF',
    buffer := subBuffer);
THIS^.processes.resetUnitController._log(
    name := 'processes.resetUnitController',
    buffer := subBuffer);
THIS^.processes.resetAlarms._log(
    name := 'processes.resetAlarms',
    buffer := subBuffer);
LOGGER(
    name := name,
    actualStatus := THIS^.actualStatus,
    previousStatus := THIS^.previousStatus,
    buffer := buffer,
    subBuffer := subBuffer,
    pHealthStatus := ADR(THIS^.statuses.healthStatus));

                
END_METHOD
END_FUNCTION_BLOCK

FUNCTION_BLOCK SM_ServicesChiller
  VAR_OUTPUT
    {attribute 'OPC.UA.DA' := '1'}
    {attribute 'OPC.UA.DA.Access' := '1'}
    actualStatus : STRING;  (* Current status description *)
    previousStatus : STRING;  (* Previous status description *)
    statuses : ServicesChillerStatuses;  (* Statuses of the state machine *)
    parts : ServicesChillerParts;  (* Parts of the state machine *)
    processes : ServicesChillerProcesses;  (* Processes of the state machine *)
  END_VAR
  VAR_IN_OUT
    {attribute 'OPC.UA.DA' := '0'}
    operatorStatus : OperatorStatus;  (* Shared operator status *)
    {attribute 'OPC.UA.DA' := '0'}
    config : ServicesChillerConfig;  (* The config *)
    {attribute 'OPC.UA.DA' := '0'}
    airTemperature : ServicesMeteoMeasurement;  (* Air temperature *)
  END_VAR

            parts.bus( isEnabled := operatorStatus.tech AND statuses.operatingStatus.manual );
parts.chillerMainController(
    isEnabled := parts.bus.isEnabled,
    config := config.chillerMainController,
    bus := parts.bus);
statuses.healthStatus(
    isGood := parts.chillerMainController.statuses.healthStatus.isGood,
    hasWarning := parts.chillerMainController.statuses.healthStatus.hasWarning);
statuses.operatingStatus();
processes.changeOperatingState( isEnabled := operatorStatus.tech );

          

{attribute 'TcRpcEnable' := '1'}
METHOD changeOperatingState : RequestResults
  VAR_INPUT
    state : OperatingStates;
  END_VAR
                  changeOperatingState := THIS^.processes.changeOperatingState.request( state := state );

                
END_METHOD

{attribute 'TcRpcEnable' := '1'}
METHOD _log : BOOL
  VAR_INPUT
    name : STRING;  (* Name of this function block instance *)
  END_VAR
  VAR_IN_OUT
    buffer : LogBuffer;  (* Buffer to write all logging to *)
  END_VAR
  VAR
    subBuffer : LogBuffer;  (* Temporary buffer to write logging by parts (sub-statemachines) to *)
  END_VAR
                  THIS^.parts.bus._log(
    name := 'bus',
    buffer := subBuffer);
THIS^.parts.chillerMainController._log(
    name := 'chillerMainController',
    buffer := subBuffer);
THIS^.processes.changeOperatingState._log(
    name := 'processes.changeOperatingState',
    buffer := subBuffer);
LOGGER(
    name := name,
    actualStatus := THIS^.actualStatus,
    previousStatus := THIS^.previousStatus,
    buffer := buffer,
    subBuffer := subBuffer,
    pHealthStatus := ADR(THIS^.statuses.healthStatus));

                
END_METHOD
END_FUNCTION_BLOCK

FUNCTION_BLOCK SM_ServicesIO
  VAR_OUTPUT
    {attribute 'OPC.UA.DA' := '1'}
    {attribute 'OPC.UA.DA.Access' := '1'}
    actualStatus : STRING;  (* Current status description *)
    previousStatus : STRING;  (* Previous status description *)
    statuses : ServicesIOStatuses;  (* Statuses of the state machine *)
    parts : ServicesIOParts;  (* Parts of the state machine *)
  END_VAR

            parts.coupler(
    id := 'COUPLER',
    typeId := 'EK1100');
parts.slot1(
    id := 'TI-RS232',
    typeId := 'EL6001');
parts.slot2(
    id := 'METEO',
    typeId := 'EL6001');
parts.slot3(
    id := 'WESTS',
    typeId := 'EL6001');
parts.slot4(
    id := 'TI-PTP',
    typeId := 'EL6688');
statuses.healthStatus( isGood := parts.coupler.statuses.healthStatus.isGood AND (parts.slot1.statuses.healthStatus.isGood AND (parts.slot2.statuses.healthStatus.isGood AND (parts.slot3.statuses.healthStatus.isGood AND parts.slot4.statuses.healthStatus.isGood))) );

          

{attribute 'TcRpcEnable' := '1'}
METHOD _log : BOOL
  VAR_INPUT
    name : STRING;  (* Name of this function block instance *)
  END_VAR
  VAR_IN_OUT
    buffer : LogBuffer;  (* Buffer to write all logging to *)
  END_VAR
  VAR
    subBuffer : LogBuffer;  (* Temporary buffer to write logging by parts (sub-statemachines) to *)
  END_VAR
                  THIS^.parts.coupler._log(
    name := 'coupler',
    buffer := subBuffer);
THIS^.parts.slot1._log(
    name := 'slot1',
    buffer := subBuffer);
THIS^.parts.slot2._log(
    name := 'slot2',
    buffer := subBuffer);
THIS^.parts.slot3._log(
    name := 'slot3',
    buffer := subBuffer);
THIS^.parts.slot4._log(
    name := 'slot4',
    buffer := subBuffer);
LOGGER(
    name := name,
    actualStatus := THIS^.actualStatus,
    previousStatus := THIS^.previousStatus,
    buffer := buffer,
    subBuffer := subBuffer,
    pHealthStatus := ADR(THIS^.statuses.healthStatus));

                
END_METHOD
END_FUNCTION_BLOCK
